(* CODESYS project 底盘控制系统.project

Project tree, tasks and I/O mapping:
  Device : AM521-0808TP/TN, Shenzhen Inovance Control Technology, version 3.5.11.50
      settings: PersistentStartAdddr = 0; PersistentStartEndAddr = 524287; Mode = 1
    application Application
      libraries: Standard, * (System); IoDrvCANopenAxis, 1.11.4.0 (Inovance); HC_CANBus, 0.1.3.0 (Inovance); Util, 3.5.11.0 (System); SM3_Drive_ETC_Inovance, 1.0.5.0 (Inovance); SysFile, * (System); SysTimeRtc, * (System); CmpLog, 3.5.5.0 (System); SysMem, 3.5.5.0 (System); CmpEventMgr, 3.5.8.0 (System); CmpApp, 3.5.11.0 (System); SysTimeCore, * (System)
      task MainTask (cyclic, interval t#4ms, priority 1) calls CANOpen_Task, main
      task CANOPEN (cyclic, interval t#10ms, priority 2) calls nothing
      program main [ST]
      DifferentialMonitor
      program CANOpen_Task [ST]
      global variables GVL
      function block FB_AckermannKinematics [ST]
      trace Trace (task MainTask): main.fbMoveFSD_Torque.FF_Torque_RR, main.fbMoveFSD_Torque.Rr_Target_rpm, main.fbMoveFSD_Torque.Rr_Actual_rpm, main.fbMoveFSD_Torque.SpeedReference, main.fbMoveFSD_Torque.TargetSpeed_kmh, main.fbMoveFSD_Torque.TorqueCmd_RR, main.fbMoveFSD_Torque.Rr_SpeedError, main.fbMoveFSD_Torque.BrakeRequest
      function block FB_SteerPositionPID [ST]
      function block FB_RearWheelVelocityPID [ST]
      function block FB_AckermannInverseKinematics [ST]
      function block FB_UDP [ST]
      function block FB_PWM [ST]
      function block FB_CAN_SCU_1 [ST]
      function block FB_MoveByYaokong [ST]
      function block FB_MoveByFSD [ST]
      function block FB_CAN_CCU [ST]
      function block test [ST]
      function block FB_CAN_VCU_SES_Req [ST]
      function block FB_CAN_BMS [ST]
      function block cantesttest [LD]
      global variables PersistentVars
      function block FB_CAN_MCU_Command [ST]
      function block FB_Depack_MotorStatus2 [ST]
      function block FB_Depack_MotorStatus1 [ST]
      function block FB_MoveControlByTorque_Yaokong [ST]
      function block FB_MoveControlByTorque_FSD [ST]
    ConfigStorage
    Resources List
    Device Diagnosis
    Network Configuration
      LocalBus Config
    HardWare Configuration
    SoftMotion General Axis Pool
    Local Bus
      GL20_2CAN : GL20 2通道CAN通信接口模块, Inovance, order no. 01440308, version 00.00.00.10
          settings: ModuleBaseInfoStruct.BusType = 10; ModuleBaseInfoStruct.RackNumber = 1; ModuleBaseInfoStruct.SlotNumber = 1; COMPort1 = 32; COMPort2 = 33; devGuid1 = 'e5bf4089-cd92-4763-8943-9d7dacf300b6'; devGuid2 = '326b6049-3dfc-42ac-adce-35d035554d5f'
          unmapped channels: RxPDO_CH, TxPDO_CH
    CAN : CAN总线, INOVANCE, version 00.00.00.10
      CAN_Port : CAN Port, Inovance, version 00.00.00.10
          settings: IsFreeCAN = False; DeviceGuid = '83de0e76-e450-4053-a235-86c09473ce3d'; DeviceName = 'GE20_CAN_485'; InterfaceNo = 1; Device = 'AM521-0808TP/TN'; Port = 4; Type = 41108
        CANopen主站 : CANopen主站, Inovance, version 00.00.00.10
            settings: COPManagerSyncStruct.SyncType = 1; COPManagerSyncStruct.SyncPeriod = 10000; COPManagerHeartbeatStruct.Enable = 1; Port NO = 4; IsPortSub = True; IsMainCAN = False; IsCANExt = True; IsLocalCAN = False
          C6049 : CANopen Slaver, Inovance, order no. 1525, version 00.00.00.10
              settings: NodeID = 3; EnableExpertSettings = 1; Error Control.SlaveHeartbeat.ProduceTime = 300; Error Control.SlaveHeartbeat.NrofConsumer = 1; VendorID = 1097; ProductNumber = 1; RevisionNumber = 131075; NrofRxPDO = 4; ValidRxPDO = 2; PdoCommuIndex = 5120; CanId = 515; TxType = 255;  = 1;  = 805306432; PdoCommuIndex = 5121; CanId = 771; TxType = 255;  = 1;  = 805371968; PdoCommuIndex = 5122; CanId = 1027; TxType = 255;  = 1;  = 805437504; PdoCommuIndex = 5123; CanId = 1283; TxType = 255;  = 1;  = 805503040; NrofTxPDO = 4; ValidTxPDO = 3; PdoCommuIndex = 6144; CanId = 387; TxType = 255; InhibitTime = 50;  = 1;  = 805568576; PdoCommuIndex = 6145; CanId = 643; TxType = 255;
                InhibitTime = 50;  = 1;  = 805634112; PdoCommuIndex = 6146; CanId = 899; TxType = 255; InhibitTime = 50;  = 1;  = 805699648; PdoCommuIndex = 6147; CanId = 1155; TxType = 255; InhibitTime = 50;  = 1;  = 805765184; SdoTimeout = 1000; NrofSDO = 31; SdoCommParam = 269877536; SdoErrHandle = 2; SdoJumptoLine = 31; SdoCommParam = 269942800; SdoCommValue = 300; SdoErrHandle = 2; SdoJumptoLine = 31; SdoCommParam = 269746208; SdoCommValue = 2147483779; SdoErrHandle = 2; SdoJumptoLine = 31; SdoCommParam = 269746208; SdoCommValue = 131; SdoErrHandle = 2; SdoJumptoLine = 31; SdoCommParam = 335544608; SdoCommValue = 2147484163; SdoErrHandle = 2; SdoJumptoLine = 31; SdoCommParam = 335610144; SdoCommValue = 2147484419; SdoErrHandle = 2; SdoJumptoLine = 31;
                SdoCommParam = 335610376; SdoCommValue = 255; SdoErrHandle = 2; SdoJumptoLine = 31; SdoCommParam = 369164296; SdoErrHandle = 2; SdoJumptoLine = 31; SdoCommParam = 369164576; SdoCommValue = 805371968; SdoErrHandle = 2; SdoJumptoLine = 31; SdoCommParam = 369164296; SdoCommValue = 1; SdoErrHandle = 2; SdoJumptoLine = 31; SdoCommParam = 335610144; SdoCommValue = 771; SdoErrHandle = 2; SdoJumptoLine = 31; SdoCommParam = 335675680; SdoCommValue = 2147484675; SdoErrHandle = 2; SdoJumptoLine = 31; SdoCommParam = 335741216; SdoCommValue = 2147484931; SdoErrHandle = 2; SdoJumptoLine = 31; SdoCommParam = 402653472; SdoCommValue = 2147484035; SdoErrHandle = 2; SdoJumptoLine = 31; SdoCommParam = 402653704; SdoCommValue = 255; SdoErrHandle = 2; SdoJumptoLine = 31; SdoCommParam = 402653968; SdoCommValue = 50; SdoErrHandle = 2; SdoJumptoLine = 31; SdoCommParam = 402654480;
                SdoErrHandle = 2; SdoJumptoLine = 31; SdoCommParam = 436207624; SdoErrHandle = 2; SdoJumptoLine = 31; SdoCommParam = 436207904; SdoCommValue = 805568576; SdoErrHandle = 2; SdoJumptoLine = 31; SdoCommParam = 436207624; SdoCommValue = 1; SdoErrHandle = 2; SdoJumptoLine = 31; SdoCommParam = 402653472; SdoCommValue = 387; SdoErrHandle = 2; SdoJumptoLine = 31; SdoCommParam = 402719008; SdoCommValue = 2147484291; SdoErrHandle = 2; SdoJumptoLine = 31; SdoCommParam = 402719240; SdoCommValue = 255; SdoErrHandle = 2; SdoJumptoLine = 31; SdoCommParam = 402719504; SdoCommValue = 50; SdoErrHandle = 2; SdoJumptoLine = 31; SdoCommParam = 402720016; SdoErrHandle = 2; SdoJumptoLine = 31; SdoCommParam = 436273160; SdoErrHandle = 2; SdoJumptoLine = 31; SdoCommParam = 436273440; SdoCommValue = 805634112; SdoErrHandle = 2; SdoJumptoLine = 31; SdoCommParam = 436273160;
                SdoCommValue = 1; SdoErrHandle = 2; SdoJumptoLine = 31; SdoCommParam = 402719008; SdoCommValue = 643; SdoErrHandle = 2; SdoJumptoLine = 31; SdoCommParam = 402784544; SdoCommValue = 2147484547; SdoErrHandle = 2; SdoJumptoLine = 31; SdoCommParam = 402850080; SdoCommValue = 2147484803; SdoErrHandle = 2; SdoJumptoLine = 31; FileName = 'C6049.eds'; FileVersion = '0x02'; FileRevision = '0x01'; EDSVersion = '4.0'; Description = 'EDS for 6049  Canopen Slave'; EDS File Path = 'D:\Asoftware\InoProShop\CODESYS\Common\AM600 Data\EdsFile\C6049.eds'; EDSVersion = 'EDLS'; VendorNumber = 1097; ProductName = 'C6049'; ProductNumber = 1; RevisionNumber = 131075; OrderCode = '60'; Baudrate = 368; SimpleBootUpSlave = 1; Granularity = 0; DynamicChannelsSupported = 0; GroupMessaging = 0; NrOfRXPDO = 4; NrOfTXPDO = 4; LSS_Supported = 0; DummyUsage = 0; SDOType = 0; SDOName = 'Set Heartbeat Consumer'; SDOType = 0; SDOName = 'Set Heartbeat Producer';
                SDOType = 0; SDOName = 'Disable Emcy COB-ID'; SDOType = 0; SDOName = 'Set Emcy COB-ID'; SDOType = 0; SDOName = 'Disable PDO'; SDOType = 0; SDOName = 'Disable PDO'; SDOType = 0; SDOName = 'Set transmission type'; SDOType = 0; SDOName = 'Clear PDO mapping'; SDOType = 0; SDOName = 'Set mapping'; SDOType = 0; SDOName = 'Set number of pdos'; SDOType = 0; SDOName = 'Set and enable COB-ID'; SDOType = 0; SDOName = 'Disable PDO'; SDOType = 0; SDOName = 'Disable PDO'; SDOType = 0; SDOName = 'Disable PDO'; SDOType = 0; SDOName = 'Set transmission type'; SDOType = 0; SDOName = 'Set inhibit time'; SDOType = 0; SDOName = 'Set event time'; SDOType = 0; SDOName = 'Clear PDO mapping'; SDOType = 0; SDOName = 'Set mapping'; SDOType = 0; SDOName = 'Set number of pdos'; SDOType = 0; SDOName = 'Set and enable COB-ID'; SDOType = 0; SDOName = 'Disable PDO';
                SDOType = 0; SDOName = 'Set transmission type'; SDOType = 0; SDOName = 'Set inhibit time'; SDOType = 0; SDOName = 'Set event time'; SDOType = 0; SDOName = 'Clear PDO mapping'; SDOType = 0; SDOName = 'Set mapping'; SDOType = 0; SDOName = 'Set number of pdos'; SDOType = 0; SDOName = 'Set and enable COB-ID'; SDOType = 0; SDOName = 'Disable PDO'; SDOType = 0; SDOName = 'Disable PDO'; Recv PDO Mapping Name.Recv PDO Mapping Name = '64 DI0'; Recv PDO Mapping Name.Recv PDO Mapping Name = '64 DI1'; Recv PDO Mapping Name.Recv PDO Mapping Name = '64 AI0'; Recv PDO Mapping Name.Recv PDO Mapping Name = '64 AI1'; Send PDO Mapping Name.Send PDO Mapping Name = '64 DO0'; Send PDO Mapping Name.Send PDO Mapping Name = '64 DO1'; Send PDO Mapping Name.Send PDO Mapping Name = '64 AO0'; Send PDO Mapping Name.Send PDO Mapping Name = '64 AO1'; Is Manual change COB-ID = 0; Is Manual change COB-ID = 0; Is Manual change COB-ID = 0; Is Manual change COB-ID = 0; Is Manual change COB-ID = 0; Is Manual change COB-ID = 0; Is Manual change COB-ID = 0; Is Manual change COB-ID = 0; MandatoryObjs = 3; Object Dictionary Item = '1000;Device Type;0x00000000;7;7;RO;0;-1;-1;-1'; Object Dictionary Item = '1001;Error Register;0x0;5;7;RO;0;-1;-1;-1'; Object Dictionary Item = '1018;Identity Object;;-1;9;;-1;4;-1;-1'; Object Dictionary Item = '1018sub0;number of entries;3;5;7;RO;0;-1;4;1'; Object Dictionary Item = '1018sub1;Vendor ID;0x00000449;7;7;RO;0;-1;-1;-1';
                Object Dictionary Item = '1018sub2;Product code;0x00000001;7;7;RO;0;-1;-1;-1'; Object Dictionary Item = '1018sub3;Revision number;0x00020003;7;7;RO;0;-1;-1;-1'; ManufacturerObjs = 9; Object Dictionary Item = '2000;Index 0x2000;;-1;9;;-1;2;-1;-1'; Object Dictionary Item = '2000sub0;Set TXPDO inhibit time;0x01;5;7;RO;0;-1;-1;-1'; Object Dictionary Item = '2000sub1;TXPDO1 inhibit time;100;5;7;RW;0;-1;-1;-1'; Object Dictionary Item = '3000;64 DI0;0;27;7;RO;1;-1;-1;-1'; Object Dictionary Item = '3001;64 DI1;0x0;27;7;RO;1;-1;-1;-1'; Object Dictionary Item = '3002;64 AI0;0;27;7;RO;1;-1;-1;-1'; Object Dictionary Item = '3003;64 AI1;0x0;27;7;RO;1;-1;-1;-1'; Object Dictionary Item = '3004;64 DO0;0x0;27;7;RWW;1;-1;-1;-1'; Object Dictionary Item = '3005;64 DO1;0x0;27;7;RWW;1;-1;-1;-1'; Object Dictionary Item = '3006;64 AO0;0x0;27;7;RWW;1;-1;-1;-1'; Object Dictionary Item = '3007;64 AO1;0x0;27;7;RWW;1;-1;-1;-1'; OptionsObjs = 20; Object Dictionary Item = '1005;COB-ID SYNC message;0x80;7;7;RW;0;-1;-1;-1'; Object Dictionary Item = '1008;Device Name;4055;9;7;CONST;0;-1;-1;-1'; Object Dictionary Item = '1016;Consumer Heartbeat time group;;-1;8;;-1;2;-1;-1'; Object Dictionary Item = '1016sub0;Number of entries;1;5;7;RO;0;-1;-1;-1'; Object Dictionary Item = '1016sub1;Consumer Heartbeat time;0;7;7;RW;0;-1;-1;-1'; Object Dictionary Item = '1017;Producer Heartbeat time group;0;6;7;RW;0;-1;-1;-1'; Object Dictionary Item = '1400;Receive PDO1 parameter;;-1;9;;-1;4;-1;-1'; Object Dictionary Item = '1400sub0;Number of entries;3;5;7;RO;0;-1;-1;-1'; Object Dictionary Item = '1400sub1;COB-ID;$NodeID + 0x200;7;7;RW;0;-1;-1;-1'; Object Dictionary Item = '1400sub2;Transmission type;255;5;7;RW;0;-1;-1;-1'; Object Dictionary Item = '1400sub3;Inhibit timer;0;5;7;RW;0;-1;-1;-1'; Object Dictionary Item = '1600;Receive PDO1 mapping;;-1;9;;-1;2;-1;-1'; Object Dictionary Item = '1600sub0;Number of mapped objects;0x1;5;7;RO;0;-1;5;0'; Object Dictionary Item = '1600sub1;1.mapped object;0x30000040;7;7;RO;0;-1;-1;-1'; Object Dictionary Item = '1401;Receive PDO2 parameter;;-1;9;;-1;4;-1;-1'; Object Dictionary Item = '1401sub0;Number of entries;3;5;7;RO;0;-1;-1;-1'; Object Dictionary Item = '1401sub1;COB-ID;$NodeID + 0x300;7;7;RW;0;-1;-1;-1'; Object Dictionary Item = '1401sub2;Transmission type;255;5;7;RW;0;-1;-1;-1'; Object Dictionary Item = '1401sub3;Inhibit timer;0;5;7;RW;0;-1;-1;-1'; Object Dictionary Item = '1601;Receive PDO2 mapping;;-1;9;;-1;2;-1;-1'; Object Dictionary Item = '1601sub0;Number of mapped objects;0x1;5;7;RO;0;-1;5;0'; Object Dictionary Item = '1601sub1;1.mapped object;0x30010040;7;7;RO;0;-1;-1;-1'; Object Dictionary Item = '1402;Receive PDO3 parameter;;-1;9;;-1;4;-1;-1'; Object Dictionary Item = '1402sub0;Number of entries;3;5;7;RO;0;-1;-1;-1'; Object Dictionary Item = '1402sub1;COB-ID;$NodeID + 0x400;7;7;RW;0;-1;-1;-1';
                Object Dictionary Item = '1402sub2;Transmission type;255;5;7;RW;0;-1;-1;-1'; Object Dictionary Item = '1402sub3;Inhibit timer;0;5;7;RW;0;-1;-1;-1'; Object Dictionary Item = '1602;Receive PDO3 mapping;;-1;9;;-1;2;-1;-1'; Object Dictionary Item = '1602sub0;Number of mapped objects;0x1;5;7;RO;0;-1;5;0'; Object Dictionary Item = '1602sub1;1.mapped object;0x30020040;7;7;RO;0;-1;-1;-1'; Object Dictionary Item = '1403;Receive PDO4 parameter;;-1;9;;-1;4;-1;-1'; Object Dictionary Item = '1403sub0;Number of entries;3;5;7;RO;0;-1;-1;-1'; Object Dictionary Item = '1403sub1;COB-ID;$NodeID + 0x500;7;7;RW;0;-1;-1;-1'; Object Dictionary Item = '1403sub2;Transmission type;255;5;7;RW;0;-1;-1;-1'; Object Dictionary Item = '1403sub3;Inhibit timer;0;5;7;RW;0;-1;-1;-1'; Object Dictionary Item = '1603;Receive PDO4 mapping;;-1;9;;-1;2;-1;-1'; Object Dictionary Item = '1603sub0;Number of mapped objects;0x1;5;7;RO;0;-1;5;0'; Object Dictionary Item = '1603sub1;1.mapped object;0x30030040;7;7;RO;0;-1;-1;-1'; Object Dictionary Item = '1800;Transmit PDO1 parameter;;-1;9;;-1;5;-1;-1'; Object Dictionary Item = '1800sub0;Number of entries;0x5;5;7;RO;0;-1;-1;-1'; Object Dictionary Item = '1800sub1;COB-ID;$NodeID + 0x180;7;7;RW;0;-1;-1;-1'; Object Dictionary Item = '1800sub2;Transmission type;255;5;7;RW;0;-1;-1;-1'; Object Dictionary Item = '1800sub3;Inhibit timer;50;6;7;RW;0;-1;-1;-1'; Object Dictionary Item = '1800sub5;Event Timer;0;27;7;RW;0;-1;65535;0'; Object Dictionary Item = '1A00;Transmit PDO1 mapping;;-1;9;;-1;2;-1;-1'; Object Dictionary Item = '1A00sub0;Number of mapped objects;0x1;5;7;RO;0;-1;4;0'; Object Dictionary Item = '1A00sub1;1.mapped object;0x30040040;7;7;RO;0;-1;-1;-1'; Object Dictionary Item = '1801;Transmit PDO2 parameter;;-1;9;;-1;5;-1;-1'; Object Dictionary Item = '1801sub0;Number of entries;0x5;5;7;RO;0;-1;-1;-1'; Object Dictionary Item = '1801sub1;COB-ID;$NodeID + 0x280;7;7;RW;0;-1;-1;-1'; Object Dictionary Item = '1801sub2;Transmission type;255;5;7;RW;0;-1;-1;-1'; Object Dictionary Item = '1801sub3;Inhibit timer;50;6;7;RW;0;-1;-1;-1'; Object Dictionary Item = '1801sub5;Event Timer;0;27;7;RW;0;-1;65535;0'; Object Dictionary Item = '1A01;Transmit PDO2 mapping;;-1;9;;-1;2;-1;-1'; Object Dictionary Item = '1A01sub0;Number of mapped objects;0x1;5;7;RO;0;-1;4;0'; Object Dictionary Item = '1A01sub1;1.mapped object;0x30050040;7;7;RO;0;-1;-1;-1'; Object Dictionary Item = '1802;Transmit PDO3 parameter;;-1;9;;-1;5;-1;-1'; Object Dictionary Item = '1802sub0;Number of entries;0x5;5;7;RO;0;-1;-1;-1'; Object Dictionary Item = '1802sub1;COB-ID;$NodeID + 0x380;7;7;RW;0;-1;-1;-1'; Object Dictionary Item = '1802sub2;Transmission type;255;5;7;RW;0;-1;-1;-1'; Object Dictionary Item = '1802sub3;Inhibit timer;50;6;7;RW;0;-1;-1;-1'; Object Dictionary Item = '1802sub5;Event Timer;0;27;7;RW;0;-1;65535;0'; Object Dictionary Item = '1A02;Transmit PDO3 mapping;;-1;9;;-1;2;-1;-1'; Object Dictionary Item = '1A02sub0;Number of mapped objects;0x1;5;7;RO;0;-1;4;0'; Object Dictionary Item = '1A02sub1;1.mapped object;0x30060040;7;7;RO;0;-1;-1;-1';
                Object Dictionary Item = '1803;Transmit PDO4 parameter;;-1;9;;-1;5;-1;-1'; Object Dictionary Item = '1803sub0;Number of entries;0x5;5;7;RO;0;-1;-1;-1'; Object Dictionary Item = '1803sub1;COB-ID;$NodeID + 0x480;7;7;RW;0;-1;-1;-1'; Object Dictionary Item = '1803sub2;Transmission type;255;5;7;RW;0;-1;-1;-1'; Object Dictionary Item = '1803sub3;Inhibit timer;50;6;7;RW;0;-1;-1;-1'; Object Dictionary Item = '1803sub5;Event Timer;0;27;7;RW;0;-1;65535;0'; Object Dictionary Item = '1A03;Transmit PDO4 mapping;;-1;9;;-1;2;-1;-1'; Object Dictionary Item = '1A03sub0;Number of mapped objects;0x1;5;7;RO;0;-1;4;0'; Object Dictionary Item = '1A03sub1;1.mapped object;0x30070040;7;7;RO;0;-1;-1;-1'
              output Application.YkqRxPDO0_data : LWORD  // 64 DI1
              input  Application.YkqTxPDO0_data : LWORD  // 64 DO0
              input  Application.Emergency_Stop : BOOL  // 64 DO0.Bit0
              input  Application.DriveByYaokong : BOOL  // 64 DO0.Bit10
              input  Application.DriveBySelf : BOOL  // 64 DO0.Bit11
              input  Application.Remote_Break : BOOL  // 64 DO0.Bit15
              input  Application.YkqTxPDO1_data : LWORD  // 64 DO1
      CAN_Port_1 : CAN Port, Inovance, version 00.00.00.10
          settings: IsFreeCAN = True; DeviceGuid = '41b44ff1-ebbe-4db4-bb20-eb005c34d964'; DeviceName = 'GL20_2CAN'; Port = 32; Type = 41090
        CAN自由协议 : CAN自由协议, Inovance, version 00.00.00.10
            settings: CANBusGeneralStruct.BusNodeID = 32; IsPortSub = True; IsLocalCAN = True; IsFreeCAN = True; DeviceTaskName = 'MainTask'; IsVirtual = True; VirtualInterface = 0; TotalChannelCount = 7; channel0.SendingMethod = False; channel0.FrameType = False; channel0.FrameFormat = False; channel0.FrameID = 361; channel0.NumberOfBytes = 8; channel0.RetransmissionInterval = 20; channel0.CycleSendingTime = 20; channel0.IOMappingParamId = 4285874176; channel1.uiChannelIndex = 1; channel1.SendingMethod = False; channel1.FrameType = False; channel1.FrameFormat = False; channel1.FrameID = 617; channel1.NumberOfBytes = 8; channel1.RetransmissionInterval = 20; channel1.CycleSendingTime = 20; channel1.IOMappingParamId = 4285874177; channel2.uiChannelIndex = 2; channel2.SendingMethod = False; channel2.FrameType = False; channel2.FrameFormat = False; channel2.FrameID = 1977; channel2.NumberOfBytes = 8; channel2.RetransmissionInterval = 5; channel2.CycleSendingTime = 10; channel2.IOMappingParamId = 4285874178; channel3.uiChannelIndex = 3; channel3.SendingMethod = False; channel3.FrameType = False; channel3.FrameFormat = False; channel3.FrameID = 256; channel3.NumberOfBytes = 8;
              channel3.RetransmissionInterval = 5; channel3.CycleSendingTime = 10; channel3.IOMappingParamId = 4285874179; channel4.uiChannelIndex = 4; channel4.SendingMethod = False; channel4.FrameType = False; channel4.FrameFormat = False; channel4.FrameID = 81; channel4.NumberOfBytes = 8; channel4.RetransmissionInterval = 5; channel4.CycleSendingTime = 10; channel4.IOMappingParamId = 4285874180; channel5.uiChannelIndex = 5; channel5.SendingMethod = False; channel5.FrameType = True; channel5.FrameFormat = False; channel5.FrameID = 285206679; channel5.NumberOfBytes = 8; channel5.RetransmissionInterval = 5; channel5.CycleSendingTime = 20; channel5.IOMappingParamId = 4285874181; channel6.uiChannelIndex = 6; channel6.SendingMethod = False; channel6.FrameType = True; channel6.FrameFormat = False; channel6.FrameID = 285205911; channel6.NumberOfBytes = 8; channel6.RetransmissionInterval = 5; channel6.CycleSendingTime = 10; channel6.IOMappingParamId = 4285874182
            input  Application.ReciveCanID : DWORD  // Receive Data.FrameID
            input  Application.ReciveCanData  // Receive Data.FrameFirstAddressArray
            output Application.CAN_SES_Req_Data_F : ARRAY [0..7] OF BYTE  // Channel0
            output Application.CAN_SES_Req_Data_R : ARRAY [0..7] OF BYTE  // Channel1
            output Application.VCU_SEB_Req_Data : ARRAY [0..7] OF BYTE  // Channel2
            output Application.main.fbMoveFSD_Torque.BMS_Send_Data : ARRAY [0..7] OF BYTE  // Channel3
            output Application.main.fbMoveFSD_Torque.CCU_CAN_Data : ARRAY [0..7] OF BYTE  // Channel4
            output Application.CAN_Motor_Cmd_RR : ARRAY [0..7] OF BYTE  // Channel5
            output Application.CAN_Motor_Cmd_RL : ARRAY [0..7] OF BYTE  // Channel6
            unmapped channels: Receive Data
      CAN_Port_2 : CAN Port, Inovance, version 00.00.00.10
          settings: IsFreeCAN = False; DeviceGuid = '41b44ff1-ebbe-4db4-bb20-eb005c34d964'; DeviceName = 'GL20_2CAN'; InterfaceNo = 1; Port = 33; Type = 41090
    Serial : 串行接口, 汇川技术股份有限公司, version 00.00.00.10
      COM : Serial Port, Inovance, version 00.00.00.10
          settings: Device = AM521-0808TP/TN; devGuid = 'e348f94f-2bae-4e83-9430-22bd03696b88'
      COM_1 : Serial Port, Inovance, version 00.00.00.10
          settings: COM = 4; Device = GE20_CAN_485; Type = 1; devGuid = '83de0e76-e450-4053-a235-86c09473ce3d'
    LocalHSIO : 本地高速IO, 汇川技术股份有限公司, version 2.0.0.0
        input  Application.IsCollisionF : BOOL  // DigitalInput.Bit0
        input  Application.IsCollisionR : BOOL  // DigitalInput.Bit1
        output Application.PDO_IO_Output0 : BOOL  // DigitalOutput.Bit0
        output Application.PDO_IO_Output1 : BOOL  // DigitalOutput.Bit1
        unmapped channels: DigitalInput, DigitalOutput
    EXP_A : 扩展卡, 汇川技术股份有限公司, version 00.00.00.10
      GE20_CAN_485 : GE20_CAN_485, Inovance, version 1.0.0.0
          settings: GE20_CAN_485 ExtCard configure.SerialAlias = 4; GE20_CAN_485 ExtCard configure.CANAlias = 4
    EXP_B : 扩展卡, 汇川技术股份有限公司, version 00.00.00.10
    HwConfiguratioinDevice : SystemConfig, Inovance, version 00.00.00.10
        settings: NetworkConfigArray.NetworkConfigArray.BusType = 10; NetworkConfigArray.NetworkConfigArray.RackSum = 1; NetworkConfigArray.NetworkConfigArray.HardwareConfigArray.HardwareConfigArray.RackNo = 1; NetworkConfigArray.NetworkConfigArray.HardwareConfigArray.HardwareConfigArray.ModuleNum = 1; EnableFun = 1
*)

// Device/Application/GVL
VAR_GLOBAL
	//遥控器参数接收
	YkqTxPDO0_data	:	ARRAY[0..7] OF BYTE;
	YkqTxPDO1_data	:	ARRAY[0..7] OF BYTE;
	YkqRxPDO0_data	:	ARRAY[0..7] OF BYTE;
	DriveBySelf		:	BOOL ;
	DriveByYaokong	:	BOOL ;
	Emergency_Stop	:	BOOL;
	Remote_Break	:	BOOL;
	
	
	

	//PDO 写入的相关数据
	//电机实际转速
    ActVel_RPM_RL   : DINT; (*  (rpm) *)
    ActVel_RPM_RR   : DINT; (*  (rpm) *)

	
	// 转向系统
     CAN_SES_Req_R : FB_CAN_VCU_SES_Req;
     CAN_SES_Req_F : FB_CAN_VCU_SES_Req;
	 CAN_SES_Req_Data_F : ARRAY[0..7] OF BYTE;
     CAN_SES_Req_Data_R : ARRAY[0..7] OF BYTE;
	 //制动系统
	 VCU_SEB_Req_Data : ARRAY[0..7] OF BYTE;
	 
	 //触边检测
	 IsCollisionF	: BOOL := FALSE;
	 IsCollisionR	: BOOL := FALSE;
	 
	 //云乐电机控制指令
	 //电机左后轮 驱动电机，CAN通道6  	 ID 10FFE597  十进制285205911
	 //电机右后轮 转向电机，CAN通道5	 ID 10FFE897  十进制285206679
	 CAN_Motor_Cmd_RR	:	ARRAY[0..7] OF BYTE;
	 CAN_Motor_Cmd_RL	:	ARRAY[0..7] OF BYTE;
	 //GCAN 212发送数据（电机指令）
	 GCAN212_Send_RR_cmd     : ARRAY[0..12] OF BYTE;
	 GCAN212_Send_RL_cmd     : ARRAY[0..12] OF BYTE;
	 GCAN212_Recive_RR_status1 : ARRAY[0..7] OF BYTE;
	 GCAN212_Recive_RR_status2 : ARRAY[0..7] OF BYTE;
	 GCAN212_Recive_RL_status1 : ARRAY[0..7] OF BYTE;
	 GCAN212_Recive_RL_status2 : ARRAY[0..7] OF BYTE;
	 
	 //自动驾驶发送控制指令，通过UDP接收
	 UDP_Re_FSD_Cmd	:	ARRAY[0..12] OF BYTE;
	 
	 
	//单、双阿克曼切换标志
	//True 是单阿克曼、FALSE是双阿克曼
	AckermanModleTransfer	:	BOOL;
	
	//CAN 总线收到的数据
	ReciveCanData	:	ARRAY[0..7] OF BYTE;
	ReciveCanID		:	DWORD;
	
	//PDO，IO信号处理，防撞条一侧为True
	PDO_IO_Output0	:	BOOL	:= TRUE;
	PDO_IO_Output1	:	BOOL	:= TRUE;
	

END_VAR

// Device/Application/PersistentVars
{attribute 'qualified_only'}
VAR_GLOBAL PERSISTENT RETAIN
END_VAR

// Device/Application/CANOpen_Task
PROGRAM CANOpen_Task
VAR
END_VAR

END_PROGRAM

// Device/Application/main
PROGRAM main
VAR

	
	fbUdp		: FB_UDP;

	fbMoveYkq	: FB_MoveByYaokong;
	fbMoveFSD	: FB_MoveByFSD;
	fbMoveYkq_Torque	:	FB_MoveControlByTorque_Yaokong;
	fbMoveFSD_Torque	:	FB_MoveControlByTorque_FSD;
	
	recvBuf     : ARRAY[0..12] OF BYTE;
	
	

	
END_VAR






fbUdp();
IF DriveBySelf THEN	
	//fbMoveFSD();
	fbMoveFSD_Torque();
	
ELSIF DriveByYaokong THEN
	//遥控器控制
	//fbMoveYkq();
	fbMoveYkq_Torque();
END_IF

END_PROGRAM

// Device/Application/FB_UDP
FUNCTION_BLOCK FB_UDP
VAR_INPUT
	//xEnable     : BOOL;               // 是否使能工作
	//sendBuf_RR_Motor_Cmd	 	: ARRAY[0..12] OF BYTE;
	//sendBuf_RL_Motor_Cmd	 	: ARRAY[0..12] OF BYTE;
END_VAR
VAR_OUTPUT
	//recvBuf     : ARRAY[0..12] OF BYTE;
	
	
END_VAR
VAR
	UDP_Peer_RR	:	UDP_Peer;
	UDP_Peer_RL	:	UDP_Peer;
	UDP_Peer_FSD	:	UDP_Peer;

	UDP_Send_RR_Motor_Cmd	:	UDP_Send;
	UDP_Send_RL_Motor_Cmd	:	UDP_Send;
	UDP_Receive_RR	:	UDP_Receive;
	UDP_Receive_RL	:	UDP_Receive;
	UDP_Receive_FSD	:	UDP_Receive;
	
	IpAddrLocal_RR	:	STRING	:= '192.168.100.210';
	PortLocal_RR	:	UINT	:= 5001;
	hPeer_RR		:	DWORD;
	IpAddrLocal_RL	:	STRING	:= '192.168.100.210';
	PortLocal_RL	:	UINT	:= 5002;
	hPeer_RL		:	DWORD;
	IpAddrLocal_FSD	:	STRING	:= '192.168.100.210';
	PortLocal_FSD	:	UINT	:= 5003;
	hPeer_FSD		:	DWORD;
	
	remoteIP_RR_Motor    : STRING(80) := '192.168.100.20';
	remotePort_RR_Motor  : UINT := 4001;
	remoteIP_RL_Motor    : STRING(80) := '192.168.100.20';
	remotePort_RL_Motor  : UINT := 4002;

	
	recvbuf_RR	: ARRAY[0..12] OF BYTE;
	recvbuf_RL	: ARRAY[0..12] OF BYTE;
	recvbuf_FSD	: ARRAY[0..12] OF BYTE;
	
	CanID_RR	: UDINT;
	CanID_RL	: UDINT;


	SendErrorID_RR		:	DWORD;
	SendErrorID_RL		:	DWORD;
	bSendDone_RR		:	BOOL;
	bSendDone_RL		:	BOOL;
	bSendBusy_RR		:	BOOL;
	bSendBusy_RL		:	BOOL;
	bRecvDone_RR 		:	BOOL;
    bRecvBusy_RR 		:	BOOL;
    bRecvDone_RL 		:	BOOL;
    bRecvBusy_RL 		:	BOOL;

	

	
	fbPWM	:	FB_PWM;
	pwm	:	BOOL;
	//rTrigSend : R_TRIG;
	PeerErrorID_RR: DWORD;
	PeerErrorID_RL: DWORD;
	
	 rTrigRecv   : R_TRIG;
	 (*-------------通信超时-------------*)
    udiLastRecvTime : UDINT := 0;      // 上一次收到UDP数据时间(ms)
    udiNowTime      : UDINT;           // 当前时间(ms)
END_VAR


// ***********RR电机*********
UDP_Peer_RR(
	xEnable:=TRUE,
	strIpAddrLocal:=IpAddrLocal_RR,
	uiPortLocal:=PortLocal_RR,
	dwErrorID =>PeerErrorID_RR);

hPeer_RR := UDP_Peer_RR.hPeer;

UDP_Receive_RR(xEnable:=TRUE,
		hPeer := hPeer_RR,
		uiSize := SIZEOF(recvbuf_RR),
		pbyData := ADR(recvbuf_RR),
		xBusy => bRecvBusy_RR,
		xDone => bRecvDone_RR
		);
		
// **********RL电机***********
UDP_Peer_RL(
	xEnable:=TRUE,
	strIpAddrLocal:=IpAddrLocal_RL,
	uiPortLocal:=PortLocal_RL,
	dwErrorID =>PeerErrorID_RL);

hPeer_RL := UDP_Peer_RL.hPeer;
UDP_Receive_RL(xEnable:=TRUE,
		hPeer := hPeer_RL,
		uiSize := SIZEOF(recvbuf_RL),
		pbyData := ADR(recvbuf_RL),
		xBusy => bRecvBusy_RL,
		xDone => bRecvDone_RL
		);

//**********接收智驾控制信号**********
UDP_Peer_FSD(
	xEnable:=TRUE,
	strIpAddrLocal:=IpAddrLocal_FSD,
	uiPortLocal:=PortLocal_FSD);
	
hPeer_FSD := UDP_Peer_FSD.hPeer;

UDP_Receive_FSD(xEnable:=TRUE,
		hPeer := hPeer_FSD,
		uiSize := SIZEOF(recvbuf_FSD),
		pbyData := ADR(recvbuf_FSD)
		);



CanID_RR :=
    SHL(BYTE_TO_UDINT(recvbuf_RR[1]),24) OR
    SHL(BYTE_TO_UDINT(recvbuf_RR[2]),16) OR
    SHL(BYTE_TO_UDINT(recvbuf_RR[3]),8)  OR
         BYTE_TO_UDINT(recvbuf_RR[4]);
CanID_RL :=
    SHL(BYTE_TO_UDINT(recvbuf_RL[1]),24) OR
    SHL(BYTE_TO_UDINT(recvbuf_RL[2]),16) OR
    SHL(BYTE_TO_UDINT(recvbuf_RL[3]),8)  OR
         BYTE_TO_UDINT(recvbuf_RL[4]);


IF CanID_RR = 16#18FFE699 THEN
	GVL.GCAN212_Recive_RR_status1[0] := recvbuf_RR[5];
    GVL.GCAN212_Recive_RR_status1[1] := recvbuf_RR[6];
    GVL.GCAN212_Recive_RR_status1[2] := recvbuf_RR[7];
    GVL.GCAN212_Recive_RR_status1[3] := recvbuf_RR[8];
    GVL.GCAN212_Recive_RR_status1[4] := recvbuf_RR[9];
    GVL.GCAN212_Recive_RR_status1[5] := recvbuf_RR[10];
    GVL.GCAN212_Recive_RR_status1[6] := recvbuf_RR[11];
    GVL.GCAN212_Recive_RR_status1[7] := recvbuf_RR[12];
ELSIF CanID_RR = 16#18FFE799 THEN
	GVL.GCAN212_Recive_RR_status2[0] := recvbuf_RR[5];
    GVL.GCAN212_Recive_RR_status2[1] := recvbuf_RR[6];
    GVL.GCAN212_Recive_RR_status2[2] := recvbuf_RR[7];
    GVL.GCAN212_Recive_RR_status2[3] := recvbuf_RR[8];
    GVL.GCAN212_Recive_RR_status2[4] := recvbuf_RR[9];
    GVL.GCAN212_Recive_RR_status2[5] := recvbuf_RR[10];
    GVL.GCAN212_Recive_RR_status2[6] := recvbuf_RR[11];
    GVL.GCAN212_Recive_RR_status2[7] := recvbuf_RR[12];
END_IF

IF CanID_RL = 16#18FFE699 THEN
	GVL.GCAN212_Recive_RL_status1[0] := recvbuf_RL[5];
    GVL.GCAN212_Recive_RL_status1[1] := recvbuf_RL[6];
    GVL.GCAN212_Recive_RL_status1[2] := recvbuf_RL[7];
    GVL.GCAN212_Recive_RL_status1[3] := recvbuf_RL[8];
    GVL.GCAN212_Recive_RL_status1[4] := recvbuf_RL[9];
    GVL.GCAN212_Recive_RL_status1[5] := recvbuf_RL[10];
    GVL.GCAN212_Recive_RL_status1[6] := recvbuf_RL[11];
    GVL.GCAN212_Recive_RL_status1[7] := recvbuf_RL[12];
ELSIF CanID_RL = 16#18FFE799 THEN
	GVL.GCAN212_Recive_RL_status2[0] := recvbuf_RL[5];
    GVL.GCAN212_Recive_RL_status2[1] := recvbuf_RL[6];
    GVL.GCAN212_Recive_RL_status2[2] := recvbuf_RL[7];
    GVL.GCAN212_Recive_RL_status2[3] := recvbuf_RL[8];
    GVL.GCAN212_Recive_RL_status2[4] := recvbuf_RL[9];
    GVL.GCAN212_Recive_RL_status2[5] := recvbuf_RL[10];
    GVL.GCAN212_Recive_RL_status2[6] := recvbuf_RL[11];
    GVL.GCAN212_Recive_RL_status2[7] := recvbuf_RL[12];
END_IF

//将接受到的智驾数据转到全局变量，便于FSD程序调用
GVL.UDP_Re_FSD_Cmd := recvbuf_FSD;

		
//发送
fbPWM(Enable:=TRUE,HalfPeriod:=T#10MS);
pwm := fbPWM.PWM;
	
UDP_Send_RR_Motor_Cmd(xExecute:=pwm,
	hPeer := hPeer_RR,
	strIpAddrDst := remoteIP_RR_Motor,
	uiPortDst := remotePort_RR_Motor,
	uiSize := SIZEOF(GVL.GCAN212_Send_RR_cmd),
	pbyData := ADR(GVL.GCAN212_Send_RR_cmd),
	udiTimeOut:=500000,
	dwErrorID => SendErrorID_RR,
	xDone	=>	bSendDone_RR,
	xBusy	=>	bSendBusy_RR
);	
UDP_Send_RL_Motor_Cmd(xExecute:=pwm,
	hPeer := hPeer_RL,
	strIpAddrDst := remoteIP_RL_Motor,
	uiPortDst := remotePort_RL_Motor,
	uiSize := SIZEOF(GVL.GCAN212_Send_RL_cmd),
	pbyData := ADR(GVL.GCAN212_Send_RL_cmd),
	udiTimeOut:=500000,
	dwErrorID => SendErrorID_RL,
	xDone	=>	bSendDone_RL,
	xBusy	=>	bSendBusy_RL
);	

(*******************************)
(* UDP通信超时检测             *)
(*******************************)

END_FUNCTION_BLOCK

// Device/Application/FB_PWM
FUNCTION_BLOCK FB_PWM
VAR_INPUT
	Enable     : BOOL := TRUE;        // 使能输出
    HalfPeriod : TIME ;     // 半周期（默认500ms -> 总周期1s）
END_VAR
VAR_OUTPUT
	PWM        : BOOL := FALSE;       // 输出的PWM布尔量
END_VAR
VAR
	tmr : TON;                        // 定时器（标准TON）
END_VAR

IF NOT Enable THEN
    PWM := FALSE;
    tmr(IN := FALSE);    // 停止并复位定时器
ELSE
    // 定时器启动：计时到达 HalfPeriod 时 tmr.Q = TRUE
    tmr(IN := TRUE, PT := HalfPeriod);

    IF tmr.Q THEN
        // 到达半周期：翻转PWM并复位定时器以开始下一半周期
        PWM := NOT PWM;
        tmr(IN := FALSE);    // 复位定时器（下一循环会再设为 TRUE 重启计时）
    END_IF
END_IF

END_FUNCTION_BLOCK

// Device/Application/FB_MoveByYaokong
(*
====================================================================
 FB 名称 : FB_MoveByYaokong
 功能说明 :
 1. 解析遥控器 CAN 数据
 2. 计算目标车速与转向角
 3. Ackermann 底盘运动学解算
 4. 转向 CAN 报文下发
 5. 驱动轮速度控制
 6. 急停 / 驻车逻辑
 7. 车辆状态回传
====================================================================
*)

FUNCTION_BLOCK FB_MoveByYaokong

//====================================================================
// 输入输出
//====================================================================
VAR_INPUT
END_VAR

VAR_OUTPUT
END_VAR


//====================================================================
// 遥控器输入相关
//====================================================================
VAR
	
	fbMotorCmd_RR		:	FB_CAN_MCU_Command;
	fbMotorCmd_RL		:	FB_CAN_MCU_Command;
    // 遥控器原始数据
    RemoteDriveRaw    : BYTE;     // 前后拨杆
    RemoteSteerRaw    : BYTE;     // 左右拨杆

    // 遥控器中位与死区
    DriveCenter       : INT := 16#7F;
    DriveDeadband     : INT := 5;

    // 遥控器解析变量
    DriveOffset       : INT;
    DriveRatio        : LREAL;
    SteeringRatio     : REAL;

    // 方向标志
    Dir_FR            : BYTE;     // 前后方向
    Dir_LR            : BYTE;     // 左右方向
END_VAR


//====================================================================
// 车辆运动控制相关
//====================================================================
VAR
    // 目标速度
    TargetSpeedMax_kmh : LREAL;
    TargetSpeed_kmh    : LREAL;
	TargetSpeed_kmhtest: LREAL;
	
    // 电机目标转速
    Rr_Speed_rpm       : LREAL;
    Rl_Speed_rpm       : LREAL;
	//电机使能标志 刹车时不使能电机
	Enable_Motor	:	BOOL  := TRUE;
	//车辆行驶档位  0:N  1:D  2:R
	RR_Shift_leavel	:	BYTE;   
	RL_Shift_leavel	:	BYTE;
	//电机驱动方式  1:速度  0:力矩
	Motor_Drive_mode_RR	:	BOOL := 1 ;
	Motor_Drive_mode_RL	:	BOOL := 1 ;
	
    // 转向角
    SteeringDeg        : REAL;
    SteeringRad        : REAL;
	
	//电机状态解包
	fbDepack_MotorStatus1_RR	:	FB_Depack_MotorStatus1;
	fbDepack_MotorStatus2_RR	:	FB_Depack_MotorStatus2;
	fbDepack_MotorStatus1_RL	:	FB_Depack_MotorStatus1;
	fbDepack_MotorStatus2_RL	:	FB_Depack_MotorStatus2;
END_VAR


//====================================================================
// 转向机构参数
//====================================================================
VAR
    // 转向机构参数
    Ls_mm              : REAL := 100.0;     // 转向节转臂长度
    Pitch_mm           : REAL := 43.692;    // 转向器线角比

    // 转向计算中间量
    RackTravel_mm      : REAL;
    SteerAngle_deg     : REAL;

    // 常量
    PI                 : REAL := 3.1415926;
END_VAR


//====================================================================
// 运动学功能块
//====================================================================
VAR
    fbKine             : FB_AckermannKinematics;
    fbInvKine          : FB_AckermannInverseKinematics;
END_VAR


//====================================================================
// 驱动器控制功能块
//====================================================================
VAR
    // 右后轮
    fbPower_RR         : MC_Power_CO;
    fbMoveVel_RR       : MC_MoveVelocity_CO;
    fbStop_RR          : MC_Stop_CO;

    // 左后轮
    fbPower_RL         : MC_Power_CO;
    fbMoveVel_RL       : MC_MoveVelocity_CO;
    fbStop_RL          : MC_Stop_CO;
END_VAR


//====================================================================
// Execute脉冲控制
//====================================================================
VAR
    // 上一次速度记录
    PreSpeed_RR        : LREAL := 0.0;
    PreSpeed_RL        : LREAL := 0.0;

    // 速度变化检测
    SpeedChanged_RR    : BOOL;
    SpeedChanged_RL    : BOOL;

    // Execute脉冲
    ExecuteMove_RR     : BOOL := FALSE;
    ExecuteMove_RL     : BOOL := FALSE;

    // 单周期保持
    PulseHold_RR       : BOOL := FALSE;
    PulseHold_RL       : BOOL := FALSE;
END_VAR


//====================================================================
// 制动与驻车系统
//====================================================================
VAR
    ParkingButton      : BOOL := FALSE;
    ParkingState       : BOOL := FALSE;

    PressureValue      : BYTE := 0;
	BrakeRequest       : BOOL := FALSE;   //<<<< 新增统一刹车请求
    rTrigBtn           : R_TRIG;
END_VAR

//====================================================================
// 电机状态反馈 UDP接收到的
//====================================================================
VAR
	RR_Motor_CanID : UDINT;
	RL_Motor_CanID : UDINT;
	
END_VAR

//====================================================================
// 减速控制
//====================================================================
VAR
	// 当前是否减速
	RR_Decelerating : BOOL;
	RL_Decelerating : BOOL;
	//速度差 = 实际速度 - 目标速度
	RR_SpeedError : REAL;
    RL_SpeedError : REAL;
	// P控制
	BrakeKp : REAL := 3;      // Nm/rpm
	
	// 最大制动力矩
	BrakeTorqueMax : REAL := 130;
	
	// 当前扭矩
	RR_BrakeTorque : REAL;
	RL_BrakeTorque : REAL;
	
	// 发送给驱动器
	RR_TorqueCmd : INT;
	RR_TorqueCmd_test : INT := -30;
	RL_TorqueCmd : INT;
	
END_VAR

//====================================================================
// 其他状态变量
//====================================================================
VAR
    Break              : BOOL := FALSE;
END_VAR

(*
====================================================================
 1. 遥控器输入解析
====================================================================
*)

TargetSpeedMax_kmh := BYTE_TO_LREAL(YkqTxPDO1_data[0]) / 10.0;


RemoteDriveRaw := YkqTxPDO1_data[1];
RemoteSteerRaw := YkqTxPDO1_data[2];

Dir_FR := RemoteDriveRaw;


(*
====================================================================
 2. 前后拨杆 -> 速度比例计算
====================================================================
*)

DriveOffset := BYTE_TO_INT(RemoteDriveRaw) - DriveCenter;

// 死区处理
IF ABS(DriveOffset) <= DriveDeadband THEN

    DriveRatio := 0.0;

ELSE

    DriveRatio :=
        INT_TO_LREAL(ABS(DriveOffset) - DriveDeadband) /
        INT_TO_LREAL(127 - DriveDeadband);

END_IF;


// 限幅
IF DriveRatio > 1.0 THEN

    DriveRatio := 1.0;

ELSIF DriveRatio < 0.0 THEN

    DriveRatio := 0.0;

END_IF;


// 最终目标速度
TargetSpeed_kmh := TargetSpeedMax_kmh * DriveRatio;

//测试
//TargetSpeed_kmh:=TargetSpeed_kmhtest;

(*
====================================================================
 3. 左右拨杆 -> 转向角计算
====================================================================
*)

// 转向方向
IF RemoteSteerRaw < 127 THEN
    Dir_LR := 1;
ELSE
    Dir_LR := 2;
END_IF;


// 比例映射
SteeringRatio := BYTE_TO_REAL(RemoteSteerRaw) / 255.0;


// 映射到车轮转角
SteeringDeg := -20.0 + (SteeringRatio * 40.0);

// //测试写死
// SteeringDeg	:= 5;
// TargetSpeed_kmh	:= 5;

// 角度 -> 弧度
SteeringRad := SteeringDeg * PI / 180.0;



(*
====================================================================
 4. 转向机构解算
====================================================================
*)

// 轮胎转角 -> 齿条位移
RackTravel_mm := Ls_mm * SteeringRad;


// 齿条位移 -> 转向电机角度
SteerAngle_deg := (RackTravel_mm / Pitch_mm) * 360.0;



(*
====================================================================
 5. 转向 CAN 报文下发
====================================================================
*)

// 前桥转向
CAN_SES_Req_F(
    Tgt_StrAngle    := SteerAngle_deg,
    Tgt_StrAngleSpd := 200,
    Veh_Spd         := 50,
    Enable          := 1
);

CAN_SES_Req_Data_F := CAN_SES_Req_F.CanData;


// 后桥转向（反向）
CAN_SES_Req_R(
    Tgt_StrAngle    := -SteerAngle_deg,
    Tgt_StrAngleSpd := 200,
    Veh_Spd         := 50,
    Enable          := 1
);

CAN_SES_Req_Data_R := CAN_SES_Req_R.CanData;



(*
====================================================================
 6. Ackermann运动学解算
====================================================================
*)

fbKine(
    v_kmh := TargetSpeed_kmh,
    delta := SteeringRad,
    Dir_LR := Dir_LR
);


// 输出轮速
Rr_Speed_rpm :=  fbKine.wRR_rpm;
Rl_Speed_rpm :=  fbKine.wRL_rpm;     // 左右电机对向安装

(*
====================================================================
 7. 行驶方向处理
====================================================================
*)
//清空刹车请求
BrakeRequest := FALSE;

IF DriveRatio < 0.0 THEN

    Rr_Speed_rpm := 0.0;
    Rl_Speed_rpm := 0.0;

    BrakeRequest := TRUE;

ELSIF DriveOffset > 0 THEN

    RR_Shift_leavel := 2;
    RL_Shift_leavel := 1;
	//RR_SpeedError := GVL.ActVel_RPM_RR - Rr_Speed_rpm;
	//RL_SpeedError := GVL.ActVel_RPM_RL - Rl_Speed_rpm;

ELSE

    RR_Shift_leavel := 1;
    RL_Shift_leavel := 2;
	//RR_SpeedError := Rr_Speed_rpm - GVL.ActVel_RPM_RR;
	//RL_SpeedError := Rl_Speed_rpm - GVL.ActVel_RPM_RL;

END_IF;

//------------------------------------------------------
// RR减速判断
//------------------------------------------------------

IF RR_SpeedError > 5 THEN

    RR_Decelerating := TRUE;

ELSIF RR_SpeedError < 1 THEN

    RR_Decelerating := FALSE;

END_IF;


//------------------------------------------------------
// RL减速判断
//------------------------------------------------------

IF RL_SpeedError > 5 THEN

    RL_Decelerating := TRUE;

ELSIF RL_SpeedError < 1 THEN

    RL_Decelerating := FALSE;

END_IF;

//------------------------------------------------------
// RR P制动
//------------------------------------------------------

IF RR_Decelerating THEN

    RR_BrakeTorque :=
        BrakeKp * RR_SpeedError;

    IF RR_BrakeTorque > BrakeTorqueMax THEN
        RR_BrakeTorque := BrakeTorqueMax;
    END_IF;

    RR_TorqueCmd :=
        -REAL_TO_INT(RR_BrakeTorque * 10);

ELSE

    RR_TorqueCmd := 0;

END_IF;


//------------------------------------------------------
// RL P制动
//------------------------------------------------------

IF RL_Decelerating THEN

    RL_BrakeTorque :=
        BrakeKp * RL_SpeedError;

    IF RL_BrakeTorque > BrakeTorqueMax THEN
        RL_BrakeTorque := BrakeTorqueMax;
    END_IF;

    RL_TorqueCmd :=
        -REAL_TO_INT(RL_BrakeTorque * 10.0);

ELSE

    RL_TorqueCmd := 0;

END_IF;




(*
====================================================================
 8. 急停逻辑
====================================================================
*)
//遥控器急停按键
IF GVL.Emergency_Stop THEN

    BrakeRequest := TRUE;

    Rr_Speed_rpm := 0.0;
    Rl_Speed_rpm := 0.0;

END_IF;

//触边传感器急停

IF GVL.IsCollisionF OR GVL.IsCollisionR THEN

    BrakeRequest := TRUE;

    Rr_Speed_rpm := 0.0;
    Rl_Speed_rpm := 0.0;

END_IF;


(*
====================================================================
 9. 驻车按键
====================================================================
*)
rTrigBtn(CLK := GVL.Remote_Break);

// 按键翻转
IF rTrigBtn.Q THEN
    ParkingState := NOT ParkingState;
END_IF;

// 驻车压力
IF ParkingState THEN

    BrakeRequest := TRUE;

    Rr_Speed_rpm := 0.0;
    Rl_Speed_rpm := 0.0;

END_IF;
(*
=========================================================
统一制动处理
=========================================================
*)

IF BrakeRequest THEN

    PressureValue := 60;

    Enable_Motor := FALSE;

    Rr_Speed_rpm := 0.0;
    Rl_Speed_rpm := 0.0;

ELSE

    PressureValue := 0;

    Enable_Motor := TRUE;

END_IF;

//====================================================================
// 切换驱动模式
//====================================================================
//RR
IF RR_Decelerating THEN
    Motor_Drive_mode_RR := FALSE;      // 扭矩模式
ELSE
    Motor_Drive_mode_RR := TRUE;       // 速度模式
END_IF;

//RL
IF RL_Decelerating THEN
    Motor_Drive_mode_RL := FALSE;
ELSE
    Motor_Drive_mode_RL := TRUE;
END_IF;

(*
====================================================================
 	下发电机控制指令
====================================================================
*)   

fbMotorCmd_RL(
	CanID := 16#10FFE597,
	Gear_Cmd := RL_Shift_leavel,
	DriveMode := Motor_Drive_mode_RL,
	MCU_Enable := Enable_Motor,
	SpeedCmd := LREAL_TO_UINT(Rl_Speed_rpm),
	TorqueCmd := RL_TorqueCmd,
	TxFrame	=> GVL.CAN_Motor_Cmd_RL,
	UdpTxFrame => GCAN212_Send_RL_cmd);
	
fbMotorCmd_RR(
	CanID := 16#10FFE597,
	Gear_Cmd := RR_Shift_leavel,
	DriveMode := Motor_Drive_mode_RR,
	MCU_Enable := Enable_Motor,
	SpeedCmd := LREAL_TO_UINT(Rr_Speed_rpm),
	TorqueCmd := RR_TorqueCmd_test,
	TxFrame	=> GVL.CAN_Motor_Cmd_RR,
	UdpTxFrame => GCAN212_Send_RR_cmd);
(*
====================================================================
 	下发制动指令
====================================================================
*)

VCU_SEB_Req_Data[0] := 6;
VCU_SEB_Req_Data[3] := PressureValue;

(*
====================================================================
 15. 底盘反解车速
====================================================================
*)

fbDepack_MotorStatus1_RL(RxData := GVL.GCAN212_Recive_RL_status1,
						 SpeedFdk => GVL.ActVel_RPM_RL);
fbDepack_MotorStatus1_RR(RxData := GVL.GCAN212_Recive_RR_status1,
						 SpeedFdk => GVL.ActVel_RPM_RR);


fbInvKine(
    ActVel_RL     :=  GVL.ActVel_RPM_RL,
    ActVel_RR     :=  GVL.ActVel_RPM_RR ,
    SteerAngle_FL := fbKine.deltaL,
    SteerAngle_FR := fbKine.deltaR,
    radius        := fbKine.radius
);



(*
====================================================================
 16. 回传遥控器 PDO 数据
====================================================================
*)
IF ReciveCanID = 16#444 THEN
	YkqRxPDO0_data[0] := ReciveCanData[6];

END_IF;


YkqRxPDO0_data[1] :=
    LREAL_TO_BYTE(fbInvKine.VehicleSpeed * 10);

END_FUNCTION_BLOCK

// Device/Application/FB_CAN_MCU_Command
FUNCTION_BLOCK FB_CAN_MCU_Command
VAR_INPUT
	CanID          : UDINT;      // CAN扩展帧ID
	//控制命令
	Gear_Cmd      : BYTE;      // 0=N 1=D 2=R
    DriveMode     : BOOL;      // FALSE=Torque  TRUE=Speed
    MCU_Enable    : BOOL;      // FALSE=Disable TRUE=Enable

    TorqueCmd     : INT;      // Nm，0.1Nm/bit，负值表示制动
    SpeedCmd      : UINT;      // rpm，1rpm/bit
END_VAR
VAR_OUTPUT
	TxFrame : ARRAY[0..7] OF BYTE;
	UdpTxFrame  : ARRAY[0..12] OF BYTE;     // GCAN212 UDP发送数据
END_VAR
VAR
	Torque_Raw: INT;
    Speed_Raw: UINT;
END_VAR

//======================================================
// Byte0：控制位
//======================================================
TxFrame[0] := 16#00;



// Bit0~1：档位
TxFrame[0] := TxFrame[0] OR UINT_TO_BYTE(Gear_Cmd AND 16#03);

// Bit2：驱动模式
IF DriveMode THEN
    TxFrame[0] := TxFrame[0] OR 16#04;
END_IF;

// Bit3：控制器使能
IF MCU_Enable THEN
    TxFrame[0] := TxFrame[0] OR 16#08;
END_IF;

//======================================================
// Byte1~2：TorqueCmd（INT16，小端）
//======================================================
Torque_Raw := REAL_TO_INT(TorqueCmd * 10.0);

TxFrame[1] := UINT_TO_BYTE(INT_TO_UINT(Torque_Raw) AND 16#00FF);
TxFrame[2] := UINT_TO_BYTE(SHR(INT_TO_UINT(Torque_Raw),8));

//======================================================
// Byte3~4：SpeedCmd（UINT16，小端）
//======================================================
Speed_Raw := SpeedCmd;

TxFrame[3] := UINT_TO_BYTE(Speed_Raw AND 16#00FF);
TxFrame[4] := UINT_TO_BYTE(SHR(Speed_Raw,8));

//======================================================
// Byte5~7：Reserve
//======================================================
TxFrame[5] := 16#00;
TxFrame[6] := 16#00;
TxFrame[7] := 16#00;


//======================================================
// GCAN212 UDP封装
//======================================================

// Byte0
// 扩展帧 + 数据帧 + UDP + DLC=8
UdpTxFrame[0] := 16#A8;

//------------------------------------------------------
// CAN ID（大端）
//------------------------------------------------------
UdpTxFrame[1] := UDINT_TO_BYTE(SHR(CanID,24) AND 16#FF);
UdpTxFrame[2] := UDINT_TO_BYTE(SHR(CanID,16) AND 16#FF);
UdpTxFrame[3] := UDINT_TO_BYTE(SHR(CanID,8)  AND 16#FF);
UdpTxFrame[4] := UDINT_TO_BYTE(CanID AND 16#FF);

//------------------------------------------------------
// CAN DATA
//------------------------------------------------------
UdpTxFrame[5]  := TxFrame[0];
UdpTxFrame[6]  := TxFrame[1];
UdpTxFrame[7]  := TxFrame[2];
UdpTxFrame[8]  := TxFrame[3];
UdpTxFrame[9]  := TxFrame[4];
UdpTxFrame[10] := TxFrame[5];
UdpTxFrame[11] := TxFrame[6];
UdpTxFrame[12] := TxFrame[7];

END_FUNCTION_BLOCK

// Device/Application/FB_Depack_MotorStatus1
FUNCTION_BLOCK FB_Depack_MotorStatus1
VAR_INPUT
    RxData : ARRAY[0..7] OF BYTE;
END_VAR

VAR_OUTPUT
    // Byte0
    Gear_State         : BYTE;      // 0=N 1=D 2=R
    DriveMode_State    : BOOL;      // FALSE=Torque TRUE=Speed
    MCU_Enable_State   : BOOL;

    // Byte1~2
    TorqueFdk_Raw      : INT;       // 原始值
    TorqueFdk          : REAL;      // Nm

    // Byte3~4
    SpeedFdk           : INT;       // rpm

    // Byte5
    MotorTemp_Raw      : BYTE;
    MotorTemp          : INT;       // ℃

    // Byte6
    ControlTemp_Raw    : BYTE;
    ControlTemp        : INT;       // ℃

    // Byte7
    ErrorCode          : BYTE;
END_VAR

VAR
    TempWord : WORD;
END_VAR

//==================== Byte0 ====================

Gear_State := RxData[0] AND 16#03;

DriveMode_State :=
    (RxData[0] AND 16#04) <> 0;

MCU_Enable_State :=
    (RxData[0] AND 16#08) <> 0;


//==================== Torque ====================

TempWord :=
    SHL(BYTE_TO_WORD(RxData[2]),8)
    OR BYTE_TO_WORD(RxData[1]);

TorqueFdk_Raw := WORD_TO_INT(TempWord);

TorqueFdk := INT_TO_REAL(TorqueFdk_Raw) * 0.1;


//==================== Speed ====================

TempWord :=
    SHL(BYTE_TO_WORD(RxData[4]),8)
    OR BYTE_TO_WORD(RxData[3]);

SpeedFdk := WORD_TO_INT(TempWord);


//==================== Temperature ====================

MotorTemp_Raw := RxData[5];
MotorTemp := BYTE_TO_INT(RxData[5]) - 40;

ControlTemp_Raw := RxData[6];
ControlTemp := BYTE_TO_INT(RxData[6]) - 40;


//==================== Error ====================

ErrorCode := RxData[7];

END_FUNCTION_BLOCK

// Device/Application/FB_Depack_MotorStatus2
FUNCTION_BLOCK FB_Depack_MotorStatus2
VAR_INPUT
	RxData : ARRAY[0..7] OF BYTE;
END_VAR
VAR_OUTPUT
	// Byte0~1
    Udc_Raw     : UINT;
    Udc         : REAL;      // V 母线电压

    // Byte2~3
    Idc_Raw     : INT;
    Idc         : REAL;      // A 母线电流

    // Byte4~5
    Iphase_Raw  : UINT;
    Iphase      : REAL;      // A  相电流有效值

    // Byte6~7
    LimitWord   : WORD;

    Limit_OverTemp            : BOOL;		//过温限功率
    Limit_MotorCurrent         : BOOL;		//电机电流限功率
    Limit_UnderVoltage         : BOOL;		//欠压限功率
    Limit_BusCurrent           : BOOL;		//母线电流限功率
    Limit_OverSpeed            : BOOL;		//转速超限限功率
    CurrentSensorFault         : BOOL;		//电流传感器异常
    BusCurrentSensorFault      : BOOL;		//母线电流传感器异常
    EncoderFault               : BOOL;		//编码器异常
    OverLoadLimit              : BOOL;		//过载限功率
    OverPowerLimit             : BOOL;		//超功率限制
END_VAR
VAR
	TempWord : WORD;
END_VAR

//==================== Udc ====================

TempWord :=
    SHL(BYTE_TO_WORD(RxData[1]),8)
    OR BYTE_TO_WORD(RxData[0]);

Udc_Raw := WORD_TO_UINT(TempWord);
Udc := UINT_TO_REAL(Udc_Raw) * 0.1;


//==================== Idc ====================

TempWord :=
    SHL(BYTE_TO_WORD(RxData[3]),8)
    OR BYTE_TO_WORD(RxData[2]);

Idc_Raw := WORD_TO_INT(TempWord);
Idc := INT_TO_REAL(Idc_Raw) * 0.1;


//==================== Iphase ====================

TempWord :=
    SHL(BYTE_TO_WORD(RxData[5]),8)
    OR BYTE_TO_WORD(RxData[4]);

Iphase_Raw := WORD_TO_UINT(TempWord);
Iphase := UINT_TO_REAL(Iphase_Raw) * 0.1;


//==================== Limit Flags ====================

LimitWord :=
    SHL(BYTE_TO_WORD(RxData[7]),8)
    OR BYTE_TO_WORD(RxData[6]);

Limit_OverTemp :=
    (LimitWord AND 16#0001) <> 0;

Limit_MotorCurrent :=
    (LimitWord AND 16#0002) <> 0;

Limit_UnderVoltage :=
    (LimitWord AND 16#0004) <> 0;

Limit_BusCurrent :=
    (LimitWord AND 16#0008) <> 0;

Limit_OverSpeed :=
    (LimitWord AND 16#0010) <> 0;

CurrentSensorFault :=
    (LimitWord AND 16#0020) <> 0;

BusCurrentSensorFault :=
    (LimitWord AND 16#0040) <> 0;

EncoderFault :=
    (LimitWord AND 16#0080) <> 0;

OverLoadLimit :=
    (LimitWord AND 16#0100) <> 0;

OverPowerLimit :=
    (LimitWord AND 16#0200) <> 0;

END_FUNCTION_BLOCK

// Device/Application/FB_AckermannKinematics
FUNCTION_BLOCK FB_AckermannKinematics
VAR_INPUT
	v_kmh		:	LREAL;	//前进速度（km/h)，车辆质心
	delta	:	LREAL;	//等效前轮转角（rad）
	Dir_LR 	: BYTE;
END_VAR
VAR_OUTPUT
	deltaL  : LREAL;  // 左前轮转角 (rad)
    deltaR  : LREAL;  // 右前轮转角 (rad)
    wRL_rpm     : LREAL;  // 左后轮角速度 (rpm)
    wRR_rpm     : LREAL;  // 右后轮角速度 (rpm)
	radius   : LREAL;   // 转弯半径
END_VAR

VAR
	v_ms   :	LREAL;	//前进速度m/s
	L   : LREAL := 1.4;   // 轴距 m
    W   : LREAL := 1.150;   // 轮距 m
    rRL : LREAL := 0.25;   // 左后轮半径 m
    rRR : LREAL := 0.25;   // 右后轮半径 m
    eps : LREAL := 1E-6;   // 防止除零
	
	
    psiDot  : LREAL;   // 偏航角速度 rad/s
    vRL     : LREAL;   // 左后轮线速度
    vRR     : LREAL;   // 右后轮线速度
	tmp 	: LREAL;
	
END_VAR



v_ms := v_kmh / 3.6;  // km/h  ->  m/s

IF ABS(delta) < eps THEN
	radius := 1.0E12;  
	psiDot := 0;
	deltaL := 0;
	deltaR := 0;
	vRL := v_ms;
	vRR := v_ms;
ELSE
	radius := ABS((L/2) / TAN(delta));  //根据自行车模型算出车体转弯半径
	psiDot := v_ms / radius;
	
	deltaL := ATAN(L/2/(radius-W/2)); // 双阿克曼，前后轮转角相同，所以只以前轮计算
	deltaR := ATAN(L/2/(radius+W/2));
	
	vRL := psiDot * SQRT( EXPT((radius - W/2),2) + EXPT(L/2,2) ); //车轮的线速度 m/s
	vRR := psiDot * SQRT( EXPT((radius + W/2),2) + EXPT(L/2,2) );
END_IF

IF Dir_LR  = 2 THEN //右转
	tmp := vRL;
	vRL := vRR;
	vRR := tmp;
END_IF

wRL_rpm := vRL / rRL * 60 / (2*3.1415926);  //车轮转速 rpm
wRR_rpm := vRR / rRR * 60 / (2*3.1415926);

END_FUNCTION_BLOCK

// Device/Application/FB_AckermannInverseKinematics
FUNCTION_BLOCK FB_AckermannInverseKinematics
VAR_INPUT
	ActVel_RL    : DINT;   // 左后轮速度反馈 rpm
    ActVel_RR    : DINT;   // 右后轮速度反馈 rpm
    SteerAngle_FL: LREAL;  // 左前轮转角 (rad)
    SteerAngle_FR: LREAL;  // 右前轮转角 (rad)
	radius		 : LREAL;   		//转弯半径
END_VAR
VAR_OUTPUT
	VehicleSpeed : REAL; // 车辆质心速度 (km/h)
	delta		: REAL;  //车轮转向角
    //HeadingAngle : LREAL; // 航向角 (rad)
END_VAR
VAR
	L	:	REAL := 1.4;  //轴距
	v_RL, v_RR   : REAL; // 后轮线速度
    v_rear       : LREAL; // 后轴平均速度
    R_L, R_R     : LREAL; // 由左右前轮计算的转弯半径
    R_avg        : LREAL; // 平均转弯半径
	
	wheelRadius  : LREAL:= 0.25;  // 车轮半径 (m)
    axleLength   : LREAL := 1.4;  // 前后轴距 (m)
    trackWidth   : LREAL := 1.150;  // 前轮轮距 (m)
	eps : LREAL := 1E-6;   // 防止除零
	
	cosL    : REAL;
    cosR    : REAL;
	delta_L     : REAL;   // 左前=左后轮转角 [rad]，正值向左转
    delta_R     : REAL;   // 右前=右后轮转角 [rad]，正值向右转
END_VAR

// ============= 逆运动学计算 =============
IF ActVel_RL < 0 THEN
	ActVel_RL := -ActVel_RL;
END_IF
IF ActVel_RR < 0 THEN
	ActVel_RR := -ActVel_RR;
END_IF
// 1. 单位换算：rpm -> m/s
v_RL := DINT_TO_REAL(ActVel_RL) / 60.0 * 2.0 * 3.14159 * wheelRadius;
v_RR := DINT_TO_REAL(ActVel_RR) / 60.0 * 2.0 * 3.14159 * wheelRadius;

delta_L := ATAN((L/2) / (radius-trackWidth/2));
delta_R := ATAN((L/2) / (radius+trackWidth/2));


// 2. 核心公式：纵向速度 = 左右后轮纵向分速平均
cosL := COS(delta_L);
cosR := COS(delta_R);
// 防止 cos 接近0时数值爆炸（极端蟹行）
IF cosL < 0.05 THEN cosL := 0.05; END_IF;
IF cosR < 0.05 THEN cosR := 0.05; END_IF;

VehicleSpeed := (v_RL * cosL + v_RR * cosR) / 2.0 * 3.6;  //km/h

delta := ATAN((L/2)/radius);

END_FUNCTION_BLOCK

// Device/Application/FB_MoveByFSD
FUNCTION_BLOCK FB_MoveByFSD
VAR_INPUT
	//recvBuf : ARRAY[0..12] OF BYTE;
	//UDP_RecvBuf     : ARRAY[0..12] OF BYTE;  //UDP接收数据
	//			:	BOOL;				//初始化标志 ，没用到
END_VAR
VAR_OUTPUT
	//UDP_SendBuf_RR_Motor_Cmd     : ARRAY[0..12] OF BYTE;		//	UDP发送数据
	//UDP_SendBuf_RL_Motor_Cmd     : ARRAY[0..12] OF BYTE;
END_VAR
VAR
(*
====================================================================
运动学功能块
====================================================================
*)
	
	fbKine			:	FB_AckermannKinematics;
	fbInvKine		:	FB_AckermannInverseKinematics;


	(* 急停释放检测 *)
    xStopState : BOOL;

(*
====================================================================
CAN协议解析
====================================================================
*)
	CAN_SCU1_Recv	:	FB_CAN_SCU_1;	//
	CAN_CCU_Send	:	FB_CAN_CCU;
	CAN_BMS_Send	:	FB_CAN_BMS;
	
(*
====================================================================
CAN接收
====================================================================
*)	
//从智驾层接收到的信号
// 	CANBus_DevRxMsg_0: CANBus_DevRxMsg;
// 	rx_enable	:	BOOL;
// 	rx_DexId	:	UINT;
// 	Rx_FilterMsg	:	CANBus_RxFilter_t;
// 	RxMsg	:	CANBus_FrameMsg_t;
// 	error_ID	:	CANBus_FBErrorType_Enum;
	
(*
====================================================================
车辆目标指令
====================================================================
*)	
	Target_ForwardWheelAngle	:	LREAL;
	Target_ReardWheelAngleMap		:	LREAL;
	Target_ReardWheelAngle		:	LREAL;
	Target_Speed	:	LREAL;

(*
====================================================================
CAN数据缓存
====================================================================
*)
	//给智驾发送的CNA数据
	BMS_Send_Data	:	ARRAY[0..7] OF BYTE;
	CCU_CAN_Data	:	ARRAY[0..7] OF BYTE;
	//检测udp接收超时
	udiNowTime      : UDINT;
    udiLastChangeTime   : UDINT;
	UDP_TimeFrame	:	UINT;
	UDP_TimeFrame_Pre	:	UINT;
	UDP_RX_Timeout	:	BOOL := FALSE;
(*
====================================================================
车轮转向角
====================================================================
*)
	Angle_RL	:	LREAL;
	Angle_RR	:	LREAL;
	Angle_FL	:	LREAL;
	Angle_FR	:	LREAL;
(*
====================================================================
车轮速度
====================================================================
*)
	Speed_RR	:	LREAL;
	Speed_RL	:	LREAL;

(*
====================================================================
整车状态
====================================================================
*)
	Vehicle_Speed	:	REAL;
	Steering_Wheel_Angle	:	REAL;
	radius   : LREAL;   // 转弯半径
	
	Vehicle_ShiftLevel	:	UINT;
	
	//电机状态解包
	fbDepack_MotorStatus1_RR	:	FB_Depack_MotorStatus1;
	fbDepack_MotorStatus2_RR	:	FB_Depack_MotorStatus2;
	fbDepack_MotorStatus1_RL	:	FB_Depack_MotorStatus1;
	fbDepack_MotorStatus2_RL	:	FB_Depack_MotorStatus2;
	
(*
====================================================================
安全状态
====================================================================
*)
   	
	//触边
	
	//刹车
	Break	:	BOOL ;
	//档位
	ShiftLevel	:	UINT;
	

(*
====================================================================
转向机构参数
====================================================================
*)
	//转向
	Ls_mm    : REAL := 100.0;   // 转向节转臂长度 (mm)
    Pitch_mm : REAL := 43.692;  // 转向器线角比 (mm/rev)

    RackTravel_mm : REAL;       // 拉杆位移
    PI            : REAL := 3.1415926;
	Ratio       : REAL;         // 归一化比例 0.0~1.0
    //SteeringDeg : REAL;         // 前轮转向角度（度）
    SteeringRad : REAL;         // 前轮转角（rad）
    SteerAngle_deg : REAL;      // 转向器目标角度（deg）
	Target_ReardWheelAngleAbs: LREAL;
    Dir_LR : BYTE;
(*
====================================================================
下发电机控制指令
====================================================================
*)	
	fbMotorCmd_RR		:	FB_CAN_MCU_Command;
	fbMotorCmd_RL		:	FB_CAN_MCU_Command;
	//车辆行驶档位  0:N  1:D  2:R
	RR_Shift_leavel	:	BYTE;   
	RL_Shift_leavel	:	BYTE;
	//电机驱动方式  1:速度  0:力矩
	Motor_Drive_mode_RR	:	BOOL := 1 ;
	Motor_Drive_mode_RL	:	BOOL := 1 ;
	Eanble_Motor	:	BOOL:=TRUE;
(*
====================================================================
制动系统相关指令
====================================================================
*)
	PressureValue	: BYTE;
	BrakeRequest : BOOL := FALSE;
	
(*
====================================================================
调试变量
====================================================================
*)	
	test : BOOL := TRUE;

	Target_SpeedTest	:	LREAL;
	Target_ReardWheelAngleTest		:	LREAL;
	
END_VAR

(*
====================================================================
 自动驾驶模式主控制逻辑
 功能：
 1. 自动驾驶初始化
 2. CAN 指令解析
 3. 底盘运动学解算
 4. 驱动轮速度控制
 5. 转向执行
 6. 急停 / 防撞 / 制动逻辑
 7. 整车状态回传
====================================================================
*)

(*
====================================================================
 0. CAN数据接收
====================================================================
*)


(*
====================================================================
 3. 自动驾驶 CAN 指令解析
====================================================================
*)
//IF ReciveCanID = 16#121 THEN

    // 解析 SCU 控制报文
    CAN_SCU1_Recv(
        RawFrame                      := GVL.UDP_Re_FSD_Cmd,
        SCU_Brk_En                    => Break,
        SCU_Target_Speed              => Target_Speed,
        SCU_Steering_Wheel_Angle_F    => Target_ReardWheelAngleMap,
		SCU_ShiftLevel_Req			  => ShiftLevel,
		Time_Frame					  => UDP_TimeFrame
    );

//END_IF;
Target_ReardWheelAngle := Target_ReardWheelAngleMap / 4.444;
IF Target_ReardWheelAngle > 20 THEN
	Target_ReardWheelAngle := 20;
ELSIF Target_ReardWheelAngle < -20 THEN
	Target_ReardWheelAngle := -20;
END_IF

//清空刹车需求
BrakeRequest := FALSE;

(*
====================================================================
 4. 底盘运动学正解
 输入：
    Target_Speed             目标车速
    Target_ReardWheelAngle   目标转角
 输出：
    左右轮转速
    左右轮转角
====================================================================
*)
//增加一个转向方向1,2
Target_ReardWheelAngleAbs := ABS(Target_ReardWheelAngle);
IF Target_ReardWheelAngle >=0 THEN
	Dir_LR := 1;
ELSE
	Dir_LR:=2;
END_IF

fbKine(
    v_kmh  := Target_Speed,
    delta  := Target_ReardWheelAngleAbs * PI / 180,
	Dir_LR := Dir_LR,
    deltaL => Angle_RL,
    deltaR => Angle_RR,

    wRL_rpm => Speed_RL,
    wRR_rpm => Speed_RR,

    radius => radius
);


(*
====================================================================
 5. 单 / 双阿克曼模式切换
====================================================================
*)
IF GVL.AckermanModleTransfer THEN

    // 单阿克曼模式
    Angle_FL := 0.0;
    Angle_FR := 0.0;

ELSE

    // 双阿克曼模式
    Angle_FL := Angle_RL;
    Angle_FR := Angle_RR;

END_IF;


(*
====================================================================
 6. 碰撞保护
====================================================================
*)
IF GVL.IsCollisionF OR GVL.IsCollisionR THEN

    BrakeRequest := TRUE;

END_IF;


(*
====================================================================
 7. 制动 / 急停保护
====================================================================
*)
xStopState := Break OR GVL.Emergency_Stop;

IF xStopState THEN

    BrakeRequest := TRUE;

END_IF;


(*
====================================================================
档位判断
0、2:空挡  1:D   2:R
====================================================================
*)

CASE ShiftLevel OF
	0:
		Speed_RR :=0;
		Speed_RL :=0;
		Vehicle_ShiftLevel := 0;
		BrakeRequest := TRUE;
		
	2:
		Speed_RR :=0;
		Speed_RL :=0;
		Vehicle_ShiftLevel:= 2;
		BrakeRequest := TRUE;
		
	1:  //前进

		RR_Shift_leavel := 2;
		RL_Shift_leavel := 1;
		Vehicle_ShiftLevel:=1;
		
		
	3:	//后退
		RR_Shift_leavel := 1;
		RL_Shift_leavel := 2;
		Vehicle_ShiftLevel:= 3;
		
ELSE
	;
END_CASE



(*
====================================================================
指令接收超时停止
====================================================================
*)
udiNowTime := SysTimeGetMs();
IF UDP_TimeFrame <> UDP_TimeFrame_Pre THEN
	UDP_TimeFrame_Pre := UDP_TimeFrame;
	udiLastChangeTime := udiNowTime;
	UDP_RX_Timeout := FALSE;
ELSE
	//判断时间
	IF  (udiNowTime - udiLastChangeTime) >= 1000 THEN
		UDP_RX_Timeout := TRUE;
	ELSE 
		UDP_RX_Timeout := FALSE;
	END_IF
END_IF


IF UDP_RX_Timeout THEN

    BrakeRequest := TRUE;

END_IF;

(*
=========================================================
统一制动处理
=========================================================
*)

IF BrakeRequest THEN

    Speed_RR := 0.0;
    Speed_RL := 0.0;

    PressureValue := 60;

    Eanble_Motor := FALSE;

ELSE

    PressureValue := 0;

    Eanble_Motor := TRUE;

END_IF;

(*
====================================================================
	下发电机控制指令
====================================================================
*)

fbMotorCmd_RR(
	CanID := 16#10FFE597,
	Gear_Cmd := RR_Shift_leavel,
	DriveMode := Motor_Drive_mode_RR,
	MCU_Enable := Eanble_Motor,
	SpeedCmd := LREAL_TO_UINT(Speed_RR),
	TxFrame	=> GVL.CAN_Motor_Cmd_RR,
	UdpTxFrame => GCAN212_Send_RR_cmd);
fbMotorCmd_RL(
	CanID := 16#10FFE597,
	Gear_Cmd := RL_Shift_leavel,
	DriveMode := Motor_Drive_mode_RL,
	MCU_Enable := Eanble_Motor,
	SpeedCmd := LREAL_TO_UINT(Speed_RL),
	TxFrame	=> GVL.CAN_Motor_Cmd_RL,
	UdpTxFrame => GCAN212_Send_RL_cmd);
(*
====================================================================
 	下发制动指令
====================================================================
*)  
VCU_SEB_Req_Data[0] := 6;
VCU_SEB_Req_Data[3] := PressureValue;
	

(*
====================================================================
 11. 转向执行
====================================================================
*)

// 角度 -> 弧度
SteeringRad :=
    Target_ReardWheelAngle * 3.1415926 / 180.0;

// 轮胎转角 -> 齿条位移
RackTravel_mm :=
    Ls_mm * SteeringRad;

// 齿条位移 -> 转向器角度
SteerAngle_deg :=
    (RackTravel_mm / Pitch_mm) * 360.0;

(*
--------------------------------------------------------------------
 前桥转向 CAN 报文
--------------------------------------------------------------------
*)
CAN_SES_Req_F(
    Tgt_StrAngle    := SteerAngle_deg,
	//Tgt_StrAngle    := 0,
    Tgt_StrAngleSpd := 200,
    Veh_Spd         := 50,
    Enable          := 1,

    CanData => CAN_SES_Req_Data_F
);


(*
--------------------------------------------------------------------
 后桥转向 CAN 报文
--------------------------------------------------------------------
*)
CAN_SES_Req_R(
    Tgt_StrAngle    := -SteerAngle_deg,
	//Tgt_StrAngle    := 0,
    Tgt_StrAngleSpd := 200,
    Veh_Spd         := 50,
    Enable          := 1,

    CanData => CAN_SES_Req_Data_R
);


(*
====================================================================
 13. 底盘运动学反解
====================================================================
*)
fbDepack_MotorStatus1_RL(RxData := GVL.GCAN212_Recive_RL_status1);
fbDepack_MotorStatus2_RL(RxData := GVL.GCAN212_Recive_RL_status2);

fbInvKine(
    ActVel_RL     :=  fbDepack_MotorStatus1_RL.SpeedFdk,
    ActVel_RR     :=  fbDepack_MotorStatus1_RR.SpeedFdk ,

    SteerAngle_FL := fbKine.deltaL,
    SteerAngle_FR := fbKine.deltaR,

    radius        := radius,

    VehicleSpeed  => Vehicle_Speed
);


(*
====================================================================
 14. 整车状态 CAN 回传
====================================================================
*)
CAN_CCU_Send(
    CCU_ShiftLevel_Sts        := Vehicle_ShiftLevel,
    CCU_P_Sts                 := GVL.Emergency_Stop OR GVL.Remote_Break OR Break,
    CCU_Ignition_Sts          := 1,
    CCU_Drive_Mode_Shift      := 0,

    Steering_Wheel_Direction  := TRUE,

    CCU_Steering_Wheel_Angle  := fbInvKine.delta,
    CCU_Vehicle_Speed         := fbInvKine.VehicleSpeed,

    CCU_Drive_Mode            := 1,

    Remote_Brake              := GVL.Remote_Break,
    Emergency_Brake           := GVL.Emergency_Stop,
    SCU_Brake_Singal          := Break,

    Left_Turn_Light_Sts       := test,
    Right_Turn_Light_Sts      := test,

    Position_Light_Sts        := test,
    LowBeam_Sts               := test,

    TxFrame => CCU_CAN_Data
);


(*
====================================================================
 15. BMS 状态转发
====================================================================
*)
IF ReciveCanID = 16#444 THEN

    CAN_BMS_Send(
		RxData := ReciveCanData,
        TxData => BMS_Send_Data
    );
	YkqRxPDO0_data[0] := ReciveCanData[6];
END_IF;
(*
====================================================================
 遥控器显示速度及电量
====================================================================
*)
YkqRxPDO0_data[1] :=
    LREAL_TO_BYTE(fbInvKine.VehicleSpeed * 10);

END_FUNCTION_BLOCK

// Device/Application/test
FUNCTION_BLOCK test
VAR_INPUT
END_VAR
VAR_OUTPUT
END_VAR
VAR
	udp : FB_UDP;
	recvBuf     : ARRAY[0..12] OF BYTE;
	sendBuf     : ARRAY[0..12] OF BYTE := [0,1,2,0,0,0,0,0,0,0,0,0];
	
END_VAR



//udp(sendBuf := sendBuf, recvBuf=>recvBuf);

END_FUNCTION_BLOCK

// Device/Application/FB_CAN_SCU_1
FUNCTION_BLOCK FB_CAN_SCU_1
VAR_INPUT
	RawFrame : ARRAY[0..12] OF BYTE;   // 13字节原始数据
	
END_VAR
VAR_OUTPUT
	SCU_ShiftLevel_Req	:	UINT;; //底盘档位状态
	SCU_Drive_Mode_Req	:	UINT;; //底盘驾驶模式状态
	SCU_Steering_Wheel_Angle_F	:	SINT; //前转向角度控制
	SCU_Steering_Wheel_Angle_R	:	SINT; //后转向角度控制
	SCU_Target_Speed	:	REAL; //速度控制
	SCU_Brk_En	:	BOOL; //刹车信号控制
	GW_Left_Turn_Light_Req	:	UINT; //左转向灯控制
	GW_Right_Turn_Light_Req	:	UINT; //右转向灯控制
	GW_Position_Light_Req	:	UINT; //刹车灯控制
	GW_LowBeam_Req	:	UINT; //近光灯控制
// 	angular_speed_flag	:	INT; //调节转向速度，只部分车型适用
// 	SCU_Brake_Force_Flag	:	BOOL; //调节EMB强度，只针对有EMB的车型
	Time_Frame	:	UINT;	//检测是否超时使用
	
END_VAR
VAR
	// 把13字节里真正的8字节CAN数据取出来（第6~13字节，即索引5~12）
    Data : ARRAY[0..7] OF BYTE;
    
    // 64位无符号整数，用于位字段提取（Intel = Little-Endian）
    Raw64 : ULINT;
    
    i : INT;
END_VAR


//============================================================
// 1. 提取真实的8字节CAN数据（跳过前5字节的长度+ID）
//============================================================
FOR i := 0 TO 7 DO
    //Data[i] := RawFrame[5 + i];
	Data[i] := GVl.UDP_Re_FSD_Cmd[5+i];
END_FOR;

Time_Frame := Data[7];

//============================================================
// 2. Little-Endian 拼成 64bit 整数（最方便做位操作）
//============================================================
Raw64 :=   (SHL(BYTE_TO_ULINT(Data[7]),56))
         OR (SHL(BYTE_TO_ULINT(Data[6]),48))
         OR (SHL(BYTE_TO_ULINT(Data[5]),40))
         OR (SHL(BYTE_TO_ULINT(Data[4]),32))
         OR (SHL(BYTE_TO_ULINT(Data[3]),24))
         OR (SHL(BYTE_TO_ULINT(Data[2]),16))
         OR (SHL(BYTE_TO_ULINT(Data[1]),8))
         OR  BYTE_TO_ULINT(Data[0]);

//============================================================
// 3. 按协议逐个提取信号（全部是 Intel/Little-Endian）
//============================================================

// Startbit 0, Len 2
SCU_ShiftLevel_Req := ULINT_TO_UINT(SHR(Raw64, 0) AND 16#03);

// Startbit 6, Len 2
SCU_Drive_Mode_Req := ULINT_TO_UINT(SHR(Raw64, 6) AND 16#03);

// Startbit 8, Len 8  → Byte1 的高8位
SCU_Steering_Wheel_Angle_F := ULINT_TO_SINT(SHR(Raw64, 8) AND 16#FF);

// Startbit 16, Len 8 → Byte2
SCU_Steering_Wheel_Angle_R := ULINT_TO_SINT(SHR(Raw64,16) AND 16#FF);

// Startbit 24, Len 9  → 跨Byte3[0..7] + Byte4[0]
SCU_Target_Speed := ULINT_TO_REAL(SHR(Raw64,24) AND 16#1FF) * 0.1;

// Startbit 33, Len 1  → Byte4 的 bit1
SCU_Brk_En := (SHR(Raw64,33) AND 16#01) = 16#01;

// Startbit 40, Len 2 → Byte5 bit0~1
GW_Left_Turn_Light_Req  := ULINT_TO_UINT(SHR(Raw64,40) AND 16#03);

// Startbit 42, Len 2 → Byte5 bit2~3
GW_Right_Turn_Light_Req := ULINT_TO_UINT(SHR(Raw64,42) AND 16#03);

// Startbit 46, Len 2 → Byte5 bit6~7
GW_Position_Light_Req   := ULINT_TO_UINT(SHR(Raw64,46) AND 16#03);

// Startbit 48, Len 2 → Byte6 bit0~1
GW_LowBeam_Req          := ULINT_TO_UINT(SHR(Raw64,48) AND 16#03);

// // Startbit 60, Len 1（有符号） → Byte7 bit4
// angular_speed_flag := IF (SHR(Raw64,60) AND 16#01)=1 THEN 1 ELSE 0; // 实际协议里是Signed，但只有0/1
// 
// // Startbit 60, Len 1（无符号） → 同样位置，另一个信号（两个信号重叠bit）
// SCU_Brake_Force_Flag := (SHR(Raw64,60) AND 16#01) = 16#01;

END_FUNCTION_BLOCK

// Device/Application/FB_CAN_CCU
FUNCTION_BLOCK FB_CAN_CCU
VAR_INPUT
	CCU_ShiftLevel_Sts         : UINT;   // 0~3   档位状态
    CCU_P_Sts                  : BOOL;   // 刹车踏板状态
    CCU_Ignition_Sts           : UINT;   // 0~3   点火状态
    CCU_Drive_Mode_Shift       : BOOL;   // 驾驶模式切换按钮
    Steering_Wheel_Direction   : BOOL;   // 前轮转向方向：TRUE=左转，FALSE=右转
    CCU_Steering_Wheel_Angle   : REAL;   // 实际角度 ° → 发送时×10（协议0.1°/LSB，120→12.0°或27°看标定）
    CCU_Vehicle_Speed          : REAL;   // km/h → 发送时×10（0.1km/h 精度）
    CCU_Drive_Mode             : UINT;   // 0~3   当前驾驶模式
    Remote_Brake               : BOOL;   // 遥控器刹车
    Emergency_Brake            : BOOL;   // 紧急制动
    SCU_Brake_Singal           : BOOL;   // 自动驾驶刹车请求
    Left_Turn_Light_Sts        : BOOL;   // 左转灯实际状态
    Right_Turn_Light_Sts       : BOOL;   // 右转灯实际状态
    Position_Light_Sts         : BOOL;   // 刹车灯状态
    LowBeam_Sts                : BOOL;   // 近光灯状态
END_VAR
VAR_OUTPUT
	TxFrame : ARRAY[0..7] OF BYTE;   // 只有数据
END_VAR
VAR
	Raw64      : ULINT := 0;
	Raw64_CAN      : ULINT := 0;
    angle_raw  : UINT;
    speed_raw  : UINT;
	
	i : INT;
    
	nibble : ULINT;
    
END_VAR

//======================================================
// 1. 按 Intel (Little-Endian) 顺序打包所有信号到 64bit
//======================================================
Raw64 := 0;  // 先清零

// bit 0~1: CCU_ShiftLevel_Sts (2 bits)
Raw64 := Raw64 OR SHL(UINT_TO_ULINT(CCU_ShiftLevel_Sts AND 16#03), 0);

// bit 2: CCU_P_Sts
IF CCU_P_Sts THEN
    Raw64 := Raw64 OR SHL(16#1, 2);
END_IF;

// bit 3~4: CCU_Ignition_Sts (2 bits)
Raw64 := Raw64 OR SHL(UINT_TO_ULINT(CCU_Ignition_Sts AND 16#03), 3);

// bit 5: CCU_Drive_Mode_Shift
IF CCU_Drive_Mode_Shift THEN
    Raw64 := Raw64 OR SHL(16#1, 5);
END_IF;

// bit 7: Steering_Wheel_Direction (左1 右0)
IF Steering_Wheel_Direction THEN
    Raw64 := Raw64 OR SHL(16#1, 7);
END_IF;

// bit 8~19: CCU_Steering_Wheel_Angle (12 bits, 0.1°/LSB)
angle_raw := REAL_TO_UINT(CCU_Steering_Wheel_Angle * 10.0);
Raw64 := Raw64 OR SHL(UINT_TO_ULINT(angle_raw AND 16#0FFF), 8);

// bit 20~28: CCU_Vehicle_Speed (9 bits, 0.1 km/h/LSB)
speed_raw := REAL_TO_UINT(CCU_Vehicle_Speed * 10.0);  // 关键：×10
Raw64 := Raw64 OR SHL(UINT_TO_ULINT(speed_raw AND 16#1FF), 20);

// bit 29~31: CCU_Drive_Mode (3 bits)
Raw64 := Raw64 OR SHL(UINT_TO_ULINT(CCU_Drive_Mode AND 16#07), 29);

// bit 32: Remote_Brake
IF Remote_Brake THEN
    Raw64 := Raw64 OR SHL(16#1, 32);
END_IF;

// bit 33: Emergency_Brake
IF Emergency_Brake THEN
    Raw64 := Raw64 OR SHL(16#1, 33);
END_IF;

// bit 34: SCU_Brake_Singal
IF SCU_Brake_Singal THEN
    Raw64 := Raw64 OR SHL(16#1, 34);
END_IF;

// bit 56: Left_Turn_Light_Sts
IF Left_Turn_Light_Sts THEN
    Raw64 := Raw64 OR SHL(16#1, 56);
END_IF;

// bit 57: Right_Turn_Light_Sts
IF Right_Turn_Light_Sts THEN
    Raw64 := Raw64 OR SHL(16#1, 57);
END_IF;

// bit 59: Position_Light_Sts (刹车灯)
IF Position_Light_Sts THEN
    Raw64 := Raw64 OR SHL(16#1, 59);
END_IF;

// bit 60: LowBeam_Sts
IF LowBeam_Sts THEN
    Raw64 := Raw64 OR SHL(16#1, 60);
END_IF;

//======================================================
// 2. 直接拆出 8 字节数据区（Intel 顺序已经是低字节在前）
//======================================================
TxFrame[0]  := ULINT_TO_BYTE(Raw64);           // Data0
TxFrame[1]  := ULINT_TO_BYTE(SHR(Raw64, 8));    // Data1
TxFrame[2]  := ULINT_TO_BYTE(SHR(Raw64, 16));   // Data2
TxFrame[3]  := ULINT_TO_BYTE(SHR(Raw64, 24));   // Data3
TxFrame[4]  := ULINT_TO_BYTE(SHR(Raw64, 32));   // Data4
TxFrame[5] := ULINT_TO_BYTE(SHR(Raw64, 40));   // Data5
TxFrame[6] := ULINT_TO_BYTE(SHR(Raw64, 48));   // Data6
TxFrame[7] := ULINT_TO_BYTE(SHR(Raw64, 56));   // Data7

//======================================================
// 3. 填充前5字节：DLC + CAN ID 0x51 (Standard Frame)
//    常见格式：Big-Endian ID，标准帧通常低字节有效
//======================================================
// TxFrame[0] := 16#08;         // DLC = 8
// 
// TxFrame[1] := 0;             // ID 高字节
// TxFrame[2] := 0;             
// TxFrame[3] := 0;             
// TxFrame[4] := 16#51;          // ID = 0x51，低字节放这里（常见做法）

END_FUNCTION_BLOCK

// Device/Application/FB_CAN_BMS
FUNCTION_BLOCK FB_CAN_BMS
VAR_INPUT
    RxData : ARRAY[0..7] OF BYTE;
END_VAR

VAR_OUTPUT
    TxData : ARRAY[0..7] OF BYTE;   // 仅仅返回CAN数据
END_VAR

VAR
    (* 原始值 *)
    VoltageRaw : UINT;
    CurrentRaw : INT;

    (* 实际值 *)
    VoltageReal : REAL;
    CurrentReal : REAL;

    (* 重新编码后的值 *)
    VoltageSend : UINT;
    CurrentSend : INT;
END_VAR

(* ============================= *)
(* 1. 解析接收到的CAN数据 *)
(* ============================= *)

(* 电压：低字节在前，高字节在后 *)
VoltageRaw := BYTE_TO_UINT(RxData[0]) OR SHL(BYTE_TO_UINT(RxData[1]), 8);

(* 电流：低字节在前，高字节在后 *)
CurrentRaw := BYTE_TO_INT(RxData[2]) OR SHL(BYTE_TO_INT(RxData[3]), 8);


(* ============================= *)
(* 2. 转换为实际物理量 *)
(* ============================= *)

(* 电压：0~4000 -> 0~400V *)
VoltageReal := UINT_TO_REAL(VoltageRaw) * 0.1;

(* 电流：0~1000 -> -500A~500A *)
CurrentReal := INT_TO_REAL(CurrentRaw) - 500.0;


(* ============================= *)
(* 3. 再重新编码 *)
(* ============================= *)


VoltageSend := REAL_TO_UINT(VoltageReal );
CurrentSend := REAL_TO_INT(CurrentReal );


(* ============================= *)
(* 4. 打包成CAN发送数据 *)
(* ============================= *)

(* 电压 *)
TxData[0] := UINT_TO_BYTE(VoltageSend AND 16#00FF);
TxData[1] := UINT_TO_BYTE(SHR(VoltageSend, 8));

(* 电流 *)
TxData[2] := INT_TO_BYTE(CurrentSend AND 16#00FF);
TxData[3] := INT_TO_BYTE(SHR(CurrentSend, 8));

(* 其余字节清零 *)
TxData[4] := RxData[6];
TxData[5] := 0;
TxData[6] := 0;
TxData[7] := 0;

END_FUNCTION_BLOCK

// Device/Application/FB_MoveControlByTorque_Yaokong
FUNCTION_BLOCK FB_MoveControlByTorque_Yaokong
//====================================================================
// 工业级双Ackermann轮毂电机底盘运动控制器 - 遥控器模式
// 版本：V2.5 (按通讯协议 + 速度斜坡 + 移除所有死区)
// 说明：遥控器及电机反馈精确，无需死区处理
//====================================================================

VAR_INPUT
END_VAR

VAR_OUTPUT
END_VAR

//====================================================================
// 遥控器输入
//====================================================================
VAR
    RemoteDriveRaw     : BYTE;
    RemoteSteerRaw     : BYTE;
    DriveCenter        : INT := 16#7F;
    DriveOffset        : INT;
    DriveRatio         : LREAL;
    SteeringRatio      : REAL;
    Dir_LR             : BYTE;
END_VAR

//====================================================================
// 车辆运动控制
//====================================================================
VAR
    TargetSpeedMax_kmh : LREAL;
    TargetSpeed_kmh    : LREAL;      // 遥控器原始目标速度
    SpeedReference     : LREAL := 0.0; // 斜坡后的参考速度
    Rr_Target_rpm      : LREAL;
    Rl_Target_rpm      : LREAL;
    Rr_Actual_rpm      : LREAL;
    Rl_Actual_rpm      : LREAL;
    Rr_SpeedError      : LREAL;
    Rl_SpeedError      : LREAL;
    Enable_Motor       : BOOL := TRUE;
    RR_Shift_leavel    : BYTE;
    RL_Shift_leavel    : BYTE;
END_VAR

//====================================================================
// 转向机构参数
//====================================================================
VAR
    Ls_mm         : REAL := 100.0;
    Pitch_mm      : REAL := 43.692;
    RackTravel_mm : REAL;
    SteerAngle_deg: REAL;
    PI_const      : REAL := 3.1415926;
    SteeringDeg   : REAL;
    SteeringRad   : REAL;
END_VAR

//====================================================================
// 运动学
//====================================================================
VAR
    fbKine   : FB_AckermannKinematics;
    fbInvKine: FB_AckermannInverseKinematics;
END_VAR

//====================================================================
// 电机控制
//====================================================================
VAR
    fbMotorCmd_RR : FB_CAN_MCU_Command;
    fbMotorCmd_RL : FB_CAN_MCU_Command;
END_VAR

//====================================================================
// PI + 前馈控制器
//====================================================================
VAR
    Kp             : LREAL := 3;
    Ki             : LREAL := 0;
    Integral_RR    : LREAL := 0.0;
    Integral_RL    : LREAL := 0.0;
    IntegralLimit  : LREAL := 70.0;
    FeedforwardGain: LREAL := 0.85;
    FF_Torque_RR   : LREAL;
    FF_Torque_RL   : LREAL;
    TotalTorque_RR : LREAL;
    TotalTorque_RL : LREAL;
    TorqueCmd_RR   : INT;
    TorqueCmd_RL   : INT;
    MaxTorque      : LREAL := 130.0;
    MinTorque      : LREAL := -130.0;
END_VAR

//====================================================================
// 速度斜坡参数（适配4ms周期）
//====================================================================
VAR
    RampUpRate     : LREAL := 5.0;    // km/h/s   可根据实际车辆微调
    RampDownRate   : LREAL := 15.0;    // km/h/s
    CycleTimeMs    : LREAL := 4.0;     // PLC实际任务周期
    d_t            : LREAL;
END_VAR

//====================================================================
// 制动与安全
//====================================================================
VAR
    BrakeRequest   : BOOL := FALSE;
    PressureValue  : BYTE := 0;
    rTrigBtn       : R_TRIG;
    ParkingState   : BOOL := FALSE;
END_VAR

//====================================================================
// 电机状态
//====================================================================
VAR
    fbDepack_MotorStatus1_RR : FB_Depack_MotorStatus1;
    fbDepack_MotorStatus1_RL : FB_Depack_MotorStatus1;
	IsReversingAndDecelerating : BOOL := FALSE;   // 正在后退减速过程
END_VAR

(*
====================================================================
 主控制逻辑
====================================================================
*)


(*
1. 遥控器解析 + 目标速度生成（已移除死区）
*)
TargetSpeedMax_kmh := BYTE_TO_LREAL(YkqTxPDO1_data[0]) / 10.0;
RemoteDriveRaw     := YkqTxPDO1_data[1];
RemoteSteerRaw     := YkqTxPDO1_data[2];

DriveOffset := BYTE_TO_INT(RemoteDriveRaw) - DriveCenter;
DriveRatio  := INT_TO_LREAL(DriveOffset) / 127.0;   // 直接线性映射，无死区

IF DriveRatio > 1.0 THEN DriveRatio := 1.0; END_IF;
IF DriveRatio < -1.0 THEN DriveRatio := -1.0; END_IF;

TargetSpeed_kmh := TargetSpeedMax_kmh * DriveRatio;  // 正值前进，负值后退

(*
2. 转向角计算
*)
IF RemoteSteerRaw < 127 THEN 
    Dir_LR := 1; 
ELSE 
    Dir_LR := 2; 
END_IF;
SteeringRatio := BYTE_TO_REAL(RemoteSteerRaw) / 255.0;
SteeringDeg   := -20.0 + (SteeringRatio * 40.0);
SteeringRad   := SteeringDeg * PI_const / 180.0;

(*
3. 转向机构 CAN 下发
*)
RackTravel_mm := Ls_mm * SteeringRad;
SteerAngle_deg := (RackTravel_mm / Pitch_mm) * 360.0;

CAN_SES_Req_F(Tgt_StrAngle := SteerAngle_deg, Tgt_StrAngleSpd := 200, Veh_Spd := 50, Enable := 1);
CAN_SES_Req_Data_F := CAN_SES_Req_F.CanData;

CAN_SES_Req_R(Tgt_StrAngle := -SteerAngle_deg, Tgt_StrAngleSpd := 200, Veh_Spd := 50, Enable := 1);
CAN_SES_Req_Data_R := CAN_SES_Req_R.CanData;

(*
4. 速度斜坡生成 (速度曲线)
*)
d_t := CycleTimeMs / 1000.0;

IF TargetSpeed_kmh > SpeedReference THEN
    SpeedReference := SpeedReference + RampUpRate * d_t;
    IF SpeedReference > TargetSpeed_kmh THEN SpeedReference := TargetSpeed_kmh; END_IF;
ELSE
    SpeedReference := SpeedReference - RampDownRate * d_t;
    IF SpeedReference < TargetSpeed_kmh THEN SpeedReference := TargetSpeed_kmh; END_IF;
END_IF;

(*
5. 运动学正解
*)
fbKine(v_kmh := SpeedReference, delta := ABS(SteeringRad), Dir_LR := Dir_LR);
Rr_Target_rpm := fbKine.wRR_rpm;
Rl_Target_rpm := fbKine.wRL_rpm;

(*
6. 读取实际转速
*)
fbDepack_MotorStatus1_RR(RxData := GVL.GCAN212_Recive_RR_status1);
fbDepack_MotorStatus1_RL(RxData := GVL.GCAN212_Recive_RL_status1);

Rr_Actual_rpm := INT_TO_LREAL(fbDepack_MotorStatus1_RR.SpeedFdk);
Rl_Actual_rpm := INT_TO_LREAL(fbDepack_MotorStatus1_RL.SpeedFdk);

//******判断是否是倒车减速******
IsReversingAndDecelerating := FALSE;
// 判断正在后退且处于减速过程
IF (SpeedReference <= 0 ) AND   // 曾经/当前在后退
   (Rr_Actual_rpm < 0) AND                               // 实际还在明显后退
   (Rr_Target_rpm> Rr_Actual_rpm) THEN                 // 目标速度 >= 当前参考速度（向0或停止靠近）
   
    IsReversingAndDecelerating := TRUE;
END_IF;

(*
7. 误差计算 + 前馈 + PI 控制
*)
Rr_SpeedError := Rr_Target_rpm - Rr_Actual_rpm;
Rl_SpeedError := Rl_Target_rpm - Rl_Actual_rpm;

FF_Torque_RR := Rr_Target_rpm * FeedforwardGain * 0.012;
FF_Torque_RL := Rl_Target_rpm * FeedforwardGain * 0.012;

Integral_RR := Integral_RR + Rr_SpeedError * Ki;
Integral_RL := Integral_RL + Rl_SpeedError * Ki;
Integral_RR := LIMIT(-IntegralLimit, Integral_RR, IntegralLimit);
Integral_RL := LIMIT(-IntegralLimit, Integral_RL, IntegralLimit);

TotalTorque_RR := FF_Torque_RR + Kp * Rr_SpeedError + Integral_RR;
TotalTorque_RL := FF_Torque_RL + Kp * Rl_SpeedError + Integral_RL;

(*
8. 档位处理 + 协议要求的扭矩符号修正
*)
IF DriveRatio > 0.0 THEN        // 前进
    RR_Shift_leavel := 2;
    RL_Shift_leavel := 1;
ELSIF DriveRatio < 0.0 THEN     // 后退
    RR_Shift_leavel := 1;
    RL_Shift_leavel := 2;
ELSIF DriveRatio = 0.0 THEN
    Integral_RR := 0;
    Integral_RL := 0;
END_IF;

// 只在「明显驱动意图」且「速度误差方向与驱动方向一致」时才强制正向力矩
// 否则让PI自然输出负力矩进行减速
IF (ABS(DriveRatio) > 0.05) AND (NOT BrakeRequest) THEN
    IF (DriveRatio > 0.0 AND Rr_SpeedError > 0.0) OR (DriveRatio < 0.0 AND Rr_SpeedError < 0.0) THEN
        TotalTorque_RR := ABS(TotalTorque_RR);
        TotalTorque_RL := ABS(TotalTorque_RL);
    END_IF;
END_IF;
//倒车减速给负值力矩
IF IsReversingAndDecelerating THEN
	TotalTorque_RR := -ABS(TotalTorque_RR);
    TotalTorque_RL := -ABS(TotalTorque_RL);
END_IF

(*
9. 安全保护
*)
BrakeRequest := FALSE;
IF GVL.Emergency_Stop OR GVL.IsCollisionF OR GVL.IsCollisionR THEN
    BrakeRequest := TRUE;
    Integral_RR := 0.0;
    Integral_RL := 0.0;
END_IF;

rTrigBtn(CLK := GVL.Remote_Break);
IF rTrigBtn.Q THEN ParkingState := NOT ParkingState; END_IF;

IF ParkingState THEN
    BrakeRequest := TRUE;
    Integral_RR := 0.0;
    Integral_RL := 0.0;
END_IF;

(*
10. 统一制动处理 + 最终限幅
*)
IF BrakeRequest THEN
    PressureValue := 60;
    Enable_Motor := FALSE;
    TorqueCmd_RR := 0;
    TorqueCmd_RL := 0;
    Integral_RR := 0.0;
    Integral_RL := 0.0;
    SpeedReference := 0.0;
ELSE
    PressureValue := 0;
    Enable_Motor := TRUE;
    
    TotalTorque_RR := LIMIT(MinTorque, TotalTorque_RR, MaxTorque);
    TotalTorque_RL := LIMIT(MinTorque, TotalTorque_RL, MaxTorque);
    

	   TorqueCmd_RR := REAL_TO_INT(TotalTorque_RR );
 	   TorqueCmd_RL := REAL_TO_INT(TotalTorque_RL );
END_IF;

(*
11. 下发电机指令（力矩模式）
*)
fbMotorCmd_RR(
    CanID := 16#10FFE597,
    Gear_Cmd := RR_Shift_leavel,
    DriveMode := FALSE,
    MCU_Enable := Enable_Motor,
    TorqueCmd := TorqueCmd_RR,
    TxFrame => GVL.CAN_Motor_Cmd_RR,
    UdpTxFrame => GVL.GCAN212_Send_RR_cmd
);

fbMotorCmd_RL(
    CanID := 16#10FFE597,
    Gear_Cmd := RL_Shift_leavel,
    DriveMode := FALSE,
    MCU_Enable := Enable_Motor,
    TorqueCmd := TorqueCmd_RL,
    TxFrame => GVL.CAN_Motor_Cmd_RL,
    UdpTxFrame => GVL.GCAN212_Send_RL_cmd
);

(*
12. 制动指令
*)
VCU_SEB_Req_Data[0] := 6;
VCU_SEB_Req_Data[3] := PressureValue;

(*
13. 车速反解与显示
*)
fbInvKine(
    ActVel_RL := fbDepack_MotorStatus1_RL.SpeedFdk,
    ActVel_RR := fbDepack_MotorStatus1_RR.SpeedFdk,
    SteerAngle_FL := fbKine.deltaL,
    SteerAngle_FR := fbKine.deltaR,
    radius := fbKine.radius
);

IF ReciveCanID = 16#444 THEN
    YkqRxPDO0_data[0] := ReciveCanData[6];
END_IF;
YkqRxPDO0_data[1] := LREAL_TO_BYTE(fbInvKine.VehicleSpeed * 10);

END_FUNCTION_BLOCK

// Device/Application/FB_MoveControlByTorque_FSD
FUNCTION_BLOCK FB_MoveControlByTorque_FSD
//====================================================================
// 工业级双Ackermann轮毂电机底盘运动控制器 - 智驾模式
// 版本：V2.1 (结构化优化版)
// 输入来源：智驾层 UDP/CAN 指令
//====================================================================

VAR_INPUT
END_VAR

VAR_OUTPUT
END_VAR
 //反馈给智驾的信息
VAR
	CAN_BMS_Send	:	FB_CAN_BMS;
	CAN_CCU_Send	:	FB_CAN_CCU;
	CCU_CAN_Data	:	ARRAY[0..7] OF BYTE;  //整车状态
	BMS_Send_Data	:	ARRAY[0..7] OF BYTE;
	
END_VAR
//====================================================================
// 智驾指令解析
//====================================================================
VAR
    CAN_SCU1_Recv     : FB_CAN_SCU_1;
    
    Target_Speed      : LREAL;
    Target_ReardWheelAngleMap : LREAL;
    Target_ReardWheelAngle : LREAL;
    ShiftLevel        : UINT := 1;
    Break             : BOOL;
    UDP_TimeFrame     : UINT;
    UDP_TimeFrame_Pre : UINT;
	IsReversingAndDecelerating: BOOL;
END_VAR

//====================================================================
// 速度指令与斜坡
//====================================================================
VAR
    TargetSpeed_kmh    : LREAL;
    SpeedReference     : LREAL;
    
    RampUpRate         : LREAL := 5.0;     // km/h/s
    RampDownRate       : LREAL := 15.0;    // km/h/s
    
END_VAR

//====================================================================
// 转向控制
//====================================================================
VAR
    Ls_mm              : REAL := 100.0;
    Pitch_mm           : REAL := 43.692;
    RackTravel_mm      : REAL;
    SteerAngle_deg     : REAL;
    PI_const           : REAL := 3.1415926;
    SteeringRad        : REAL;
    Target_ReardWheelAngleAbs : LREAL;
    Dir_LR             : BYTE;
END_VAR

//====================================================================
// 运动学
//====================================================================
VAR
    fbKine             : FB_AckermannKinematics;
    fbInvKine          : FB_AckermannInverseKinematics;
END_VAR

//====================================================================
// 电机反馈与状态
//====================================================================
VAR
    Rr_Target_rpm      : LREAL;
    Rl_Target_rpm      : LREAL;
    Rr_Actual_rpm      : LREAL;
    Rl_Actual_rpm      : LREAL;
    Rr_SpeedError      : LREAL;
    Rl_SpeedError      : LREAL;
    
    fbDepack_MotorStatus1_RR : FB_Depack_MotorStatus1;
    fbDepack_MotorStatus1_RL : FB_Depack_MotorStatus1;
END_VAR

//====================================================================
// PI + 前馈 控制器
//====================================================================
VAR
    Kp                 : LREAL := 4;
    Ki                 : LREAL := 0;
    Integral_RR        : LREAL := 0.0;
    Integral_RL        : LREAL := 0.0;
    IntegralLimit      : LREAL := 65.0;
    
    FeedforwardGain    : LREAL := 0.72;
    FF_Torque_RR       : LREAL;
    FF_Torque_RL       : LREAL;
    
    TotalTorque_RR     : LREAL;
    TotalTorque_RL     : LREAL;
    TorqueCmd_RR       : INT;
    TorqueCmd_RL       : INT;
    
    MaxTorque          : LREAL := 130.0;
    MinTorque          : LREAL := -130.0;
END_VAR

//====================================================================
// 停车与零速逻辑
//====================================================================
VAR
    BrakeRequest       : BOOL := FALSE;
    PressureValue      : BYTE := 0;
    Enable_Motor       : BOOL := TRUE;
    
    RR_Shift_leavel    : BYTE;
    RL_Shift_leavel    : BYTE;
    
    // 超时检测
    udiNowTime         : UDINT;
    udiLastChangeTime  : UDINT;
    UDP_RX_Timeout     : BOOL := FALSE;
END_VAR

//====================================================================
// 安全
//====================================================================
VAR
    Vehicle_ShiftLevel : UINT;
END_VAR

//====================================================================
// 电机控制
//====================================================================
VAR
    fbMotorCmd_RR      : FB_CAN_MCU_Command;
    fbMotorCmd_RL      : FB_CAN_MCU_Command;
END_VAR

//====================================================================
// 循环时间
//====================================================================
VAR
    CycleTimeMs        : LREAL := 4.0;
    d_t                 : LREAL;
END_VAR

//====================================================================
// 调试变量
//====================================================================
VAR
    Target_Speed_test : LREAL;
	Target_ReardWheelAngle_test : LREAL;
END_VAR

(*
====================================================================
 主控制循环 - 智驾模式
====================================================================
*)

(*
====================================================
1. 智驾指令解析 (CAN_SCU1)
====================================================
*)
CAN_SCU1_Recv(
    //RawFrame                      := GVL.UDP_Re_FSD_Cmd,
    SCU_Brk_En                    => Break,
    SCU_Target_Speed              => Target_Speed,
    SCU_Steering_Wheel_Angle_F    => Target_ReardWheelAngleMap,
    SCU_ShiftLevel_Req            => ShiftLevel,
    Time_Frame                    => UDP_TimeFrame
);
IF Target_Speed > 5 THEN
	Target_Speed := 5;
END_IF

Target_ReardWheelAngle := Target_ReardWheelAngleMap / 4.444;
IF Target_ReardWheelAngle > 20 THEN
    Target_ReardWheelAngle := 20;
ELSIF Target_ReardWheelAngle < -20 THEN
    Target_ReardWheelAngle := -20;
END_IF;
(*
====================================================
10. 档位判断
====================================================
*)
//测试
//TargetSpeed_kmh := Target_Speed_test;
//ShiftLevel := 1;
CASE ShiftLevel OF
    1:  // 前进
		TargetSpeed_kmh := Target_Speed;
        RR_Shift_leavel := 2;
        RL_Shift_leavel := 1;
        Vehicle_ShiftLevel := 1;
    3:  // 后退
		TargetSpeed_kmh := -Target_Speed;
        RR_Shift_leavel := 1;
        RL_Shift_leavel := 2;
        Vehicle_ShiftLevel := 3;
ELSE
    ;
END_CASE;



(*
====================================================
2. 指令超时检测
====================================================
*)
udiNowTime := SysTimeGetMs();
IF UDP_TimeFrame <> UDP_TimeFrame_Pre THEN
    UDP_TimeFrame_Pre := UDP_TimeFrame;
    udiLastChangeTime := udiNowTime;
    UDP_RX_Timeout := FALSE;
ELSE
    IF (udiNowTime - udiLastChangeTime) >= 1000 THEN
        UDP_RX_Timeout := TRUE;
    ELSE 
        UDP_RX_Timeout := FALSE;
    END_IF;
END_IF;

(*
====================================================
3. 速度斜坡生成
====================================================
*)
d_t := CycleTimeMs / 1000.0;

IF TargetSpeed_kmh > SpeedReference THEN
    SpeedReference := SpeedReference + RampUpRate * d_t;
    IF SpeedReference > TargetSpeed_kmh THEN SpeedReference := TargetSpeed_kmh; END_IF;
ELSE
    SpeedReference := SpeedReference - RampDownRate * d_t;
    IF SpeedReference < TargetSpeed_kmh THEN SpeedReference := TargetSpeed_kmh; END_IF;
END_IF;


(*
====================================================
5. 转向计算与CAN下发
====================================================
*)
//测试
//Target_ReardWheelAngle := Target_ReardWheelAngle_test;
Target_ReardWheelAngleAbs := ABS(Target_ReardWheelAngle);

IF Target_ReardWheelAngle >= 0 THEN
    Dir_LR := 1;
ELSE
    Dir_LR := 2;
END_IF;

SteeringRad := Target_ReardWheelAngle * PI_const / 180.0;

RackTravel_mm := Ls_mm * SteeringRad;
SteerAngle_deg := (RackTravel_mm / Pitch_mm) * 360.0;

CAN_SES_Req_F(Tgt_StrAngle := SteerAngle_deg, Tgt_StrAngleSpd := 200, Veh_Spd := 50, Enable := 1);
CAN_SES_Req_Data_F := CAN_SES_Req_F.CanData;

CAN_SES_Req_R(Tgt_StrAngle := -SteerAngle_deg, Tgt_StrAngleSpd := 200, Veh_Spd := 50, Enable := 1);
CAN_SES_Req_Data_R := CAN_SES_Req_R.CanData;

(*
====================================================
6. Ackermann运动学正解
====================================================
*)
fbKine(v_kmh := SpeedReference, delta := ABS(SteeringRad), Dir_LR := Dir_LR);

Rr_Target_rpm := fbKine.wRR_rpm;
Rl_Target_rpm := fbKine.wRL_rpm;

(*
====================================================
7. 电机反馈读取
====================================================
*)
fbDepack_MotorStatus1_RR(RxData := GVL.GCAN212_Recive_RR_status1);
fbDepack_MotorStatus1_RL(RxData := GVL.GCAN212_Recive_RL_status1);

Rr_Actual_rpm := INT_TO_LREAL(fbDepack_MotorStatus1_RR.SpeedFdk);
Rl_Actual_rpm := INT_TO_LREAL(fbDepack_MotorStatus1_RL.SpeedFdk);

//******判断是否是倒车减速******
IsReversingAndDecelerating := FALSE;
// 判断正在后退且处于减速过程
IF (SpeedReference <= 0 ) AND   // 曾经/当前在后退
   (Rr_Actual_rpm < 0) AND                               // 实际还在明显后退
   (Rr_Target_rpm> Rr_Actual_rpm) THEN                 // 目标速度 >= 当前参考速度（向0或停止靠近）
   
    IsReversingAndDecelerating := TRUE;
END_IF;


(*
7. 误差计算 + 前馈 + PI 控制
*)
Rr_SpeedError := Rr_Target_rpm - Rr_Actual_rpm;
Rl_SpeedError := Rl_Target_rpm - Rl_Actual_rpm;

FF_Torque_RR := Rr_Target_rpm * FeedforwardGain * 0.012;
FF_Torque_RL := Rl_Target_rpm * FeedforwardGain * 0.012;

Integral_RR := Integral_RR + Rr_SpeedError * Ki;
Integral_RL := Integral_RL + Rl_SpeedError * Ki;
Integral_RR := LIMIT(-IntegralLimit, Integral_RR, IntegralLimit);
Integral_RL := LIMIT(-IntegralLimit, Integral_RL, IntegralLimit);

TotalTorque_RR := FF_Torque_RR + Kp * Rr_SpeedError + Integral_RR;
TotalTorque_RL := FF_Torque_RL + Kp * Rl_SpeedError + Integral_RL;


//倒车减速给负值力矩  否则给正力矩
IF IsReversingAndDecelerating  THEN
	TotalTorque_RR := -ABS(TotalTorque_RR);
    TotalTorque_RL := -ABS(TotalTorque_RL);
	
END_IF

(*
====================================================
9. 档位与安全制动
====================================================
*)

BrakeRequest := FALSE;
// IF Break OR UDP_RX_Timeout OR GVL.Emergency_Stop OR GVL.IsCollisionF OR GVL.IsCollisionR THEN
//     BrakeRequest := TRUE;
// END_IF;
IF Break OR GVL.Emergency_Stop OR GVL.IsCollisionF OR GVL.IsCollisionR THEN
    BrakeRequest := TRUE;
END_IF;

IF BrakeRequest THEN
    PressureValue := 60;
    Enable_Motor := FALSE;
    TorqueCmd_RR := 0;
    TorqueCmd_RL := 0;
    Integral_RR := 0.0;
    Integral_RL := 0.0;
    SpeedReference := 0.0;
ELSE
    PressureValue := 0;
    Enable_Motor := TRUE;
	TotalTorque_RR := LIMIT(MinTorque, TotalTorque_RR, MaxTorque);
    TotalTorque_RL := LIMIT(MinTorque, TotalTorque_RL, MaxTorque);
    
	TorqueCmd_RR := REAL_TO_INT(TotalTorque_RR );
 	TorqueCmd_RL := REAL_TO_INT(TotalTorque_RL );
END_IF;

(*
====================================================
11. 电机指令下发
====================================================
*)
fbMotorCmd_RR(
    CanID := 16#10FFE597,
    Gear_Cmd := RR_Shift_leavel,
    DriveMode := FALSE,
    MCU_Enable := Enable_Motor,
    TorqueCmd := TorqueCmd_RR,
    TxFrame => GVL.CAN_Motor_Cmd_RR,
    UdpTxFrame => GVL.GCAN212_Send_RR_cmd
);

fbMotorCmd_RL(
    CanID := 16#10FFE597,
    Gear_Cmd := RL_Shift_leavel,
    DriveMode := FALSE,
    MCU_Enable := Enable_Motor,
    TorqueCmd := TorqueCmd_RL,
    TxFrame => GVL.CAN_Motor_Cmd_RL,
    UdpTxFrame => GVL.GCAN212_Send_RL_cmd
);

(*
====================================================
12. 制动指令
====================================================
*)
VCU_SEB_Req_Data[0] := 6;
VCU_SEB_Req_Data[3] := PressureValue;

(*
====================================================
13. 车速反解与显示
====================================================
*)
fbInvKine(
    ActVel_RL := fbDepack_MotorStatus1_RL.SpeedFdk,
    ActVel_RR := fbDepack_MotorStatus1_RR.SpeedFdk,
    SteerAngle_FL := fbKine.deltaL,
    SteerAngle_FR := fbKine.deltaR,
    radius := fbKine.radius
);
(*
====================================================================
 14. 整车状态 CAN 回传
====================================================================
*)
CAN_CCU_Send(
    CCU_ShiftLevel_Sts        := Vehicle_ShiftLevel,
    CCU_P_Sts                 := GVL.Emergency_Stop OR GVL.Remote_Break OR Break,
    CCU_Ignition_Sts          := 1,
    CCU_Drive_Mode_Shift      := 0,

    Steering_Wheel_Direction  := TRUE,

    CCU_Steering_Wheel_Angle  := fbInvKine.delta * 4.44 * 180 / 3.1415926,
    CCU_Vehicle_Speed         := fbInvKine.VehicleSpeed,

    CCU_Drive_Mode            := 0,

    Remote_Brake              := GVL.Remote_Break,
    Emergency_Brake           := GVL.Emergency_Stop,
    SCU_Brake_Singal          := Break,

    Left_Turn_Light_Sts       := 0,
    Right_Turn_Light_Sts      := 0,

    Position_Light_Sts        := 0,
    LowBeam_Sts               := 0,

    TxFrame => CCU_CAN_Data
);

(*
====================================================================
 15. BMS 状态转发
====================================================================
*)
IF ReciveCanID = 16#444 THEN

    CAN_BMS_Send(
		RxData := ReciveCanData,
        TxData => BMS_Send_Data
    );
	YkqRxPDO0_data[0] := ReciveCanData[6];
END_IF;

YkqRxPDO0_data[1] := LREAL_TO_BYTE(fbInvKine.VehicleSpeed * 10);

END_FUNCTION_BLOCK

// Device/Application/FB_SteerPositionPID
FUNCTION_BLOCK FB_SteerPositionPID
VAR_INPUT
    deltaL_ref    : LREAL;   // 期望左前轮角度 (rad)
    deltaR_ref    : LREAL;   // 期望右前轮角度 (rad)
    dt_           : LREAL := 0.01; // 控制周期 (s)
    Kp            : LREAL := 8.0;
    Ki            : LREAL := 1.0;
    Kd            : LREAL := 0.1;
    outMax        : LREAL := 1000.0;  // 速度模式输出上限 (rpm 等)
    outMin        : LREAL := -1000.0;
    derivTau      : LREAL := 0.02;
    usePositionSetpoint : BOOL := TRUE; // TRUE: 下发位置 setpoint(TRUE：位置模式； FALSE：速度模式)
    PosUnitPerRad : LREAL := 180.0/3.14159265358979323846; // 默认 deg/rad，若你的驱动用 counts 把这里改为 counts_per_rad
    VelUnitPerRadSecToPDO : LREAL := 60.0/(2.0*3.14159265358979323846); // rad/s -> rpm
END_VAR

VAR_IN_OUT
    ActPos_FL     : DINT;   // 
    ActPos_FR     : DINT;   // 
END_VAR

VAR_OUTPUT
    PDO_TargetPos_FL : DINT; //
    PDO_TargetPos_FR : DINT;
    PDO_TargetVel_FL : DINT; // 
    PDO_TargetVel_FR : DINT;
END_VAR

VAR
    actPosRadL   : LREAL;
    actPosRadR   : LREAL;
    errL, errR   : LREAL;
    prevErrL     : LREAL := 0.0;
    prevErrR     : LREAL := 0.0;
    integralL    : LREAL := 0.0;
    integralR    : LREAL := 0.0;
    derivL_filt  : LREAL := 0.0;
    derivR_filt  : LREAL := 0.0;
    alpha        : LREAL;
    deriv_rawL   : LREAL;
    deriv_rawR   : LREAL;
    pidOutL      : LREAL; // 若输出速度则单位为 rad/s (需乘 conversion)
    pidOutR      : LREAL;
    PI_CONST     : LREAL := 3.14159265358979323846;
END_VAR

IF dt_ <= 0.0 THEN dt_ := 0.01; END_IF
alpha := derivTau / (derivTau + dt_);

(* 将 ActPos (DINT, PDO units) 转为弧度 *)
actPosRadL := DINT_TO_LREAL(ActPos_FL) / PosUnitPerRad; 
actPosRadR := DINT_TO_LREAL(ActPos_FR) / PosUnitPerRad; 

(* 位置环 PID（rad 域） *)
errL := deltaL_ref - actPosRadL;
integralL := integralL + errL * dt_;
deriv_rawL := (errL - prevErrL) / dt_;
derivL_filt := alpha * derivL_filt + (1.0 - alpha) * deriv_rawL;
pidOutL := Kp * errL + Ki * integralL + Kd * derivL_filt;

IF pidOutL > outMax THEN
    pidOutL := outMax;
    integralL := integralL - errL * dt_;
ELSIF pidOutL < outMin THEN
    pidOutL := outMin;
    integralL := integralL - errL * dt_;
END_IF
prevErrL := errL;

errR := deltaR_ref - actPosRadR;
integralR := integralR + errR * dt_;
deriv_rawR := (errR - prevErrR) / dt_;
derivR_filt := alpha * derivR_filt + (1.0 - alpha) * deriv_rawR;
pidOutR := Kp * errR + Ki * integralR + Kd * derivR_filt;

IF pidOutR > outMax THEN
    pidOutR := outMax;
    integralR := integralR - errR * dt_;
ELSIF pidOutR < outMin THEN
    pidOutR := outMin;
    integralR := integralR - errR * dt_;
END_IF
prevErrR := errR;

(* 输出 *)
IF usePositionSetpoint THEN
    (* 位置模式：把目标角（rad）转换为 PDO 单位 (PosUnitPerRad)，然后 LREAL->DINT *)
    PDO_TargetPos_FL := LREAL_TO_DINT( deltaL_ref * PosUnitPerRad );  
    PDO_TargetPos_FR := LREAL_TO_DINT( deltaR_ref * PosUnitPerRad );  
    PDO_TargetVel_FL := 0;
    PDO_TargetVel_FR := 0;
ELSE
    (* 速度模式：把 pidOut (rad/s) 转换为 PDO 速度单位 (rpm) *)
    (* 先把 pidOut（rad/s）乘以系数转换为 rpm，再 LREAL->DINT *)
    PDO_TargetVel_FL := LREAL_TO_DINT( pidOutL * VelUnitPerRadSecToPDO ); 
    PDO_TargetVel_FR := LREAL_TO_DINT( pidOutR * VelUnitPerRadSecToPDO ); 
    PDO_TargetPos_FL := 0;
    PDO_TargetPos_FR := 0;
END_IF

END_FUNCTION_BLOCK

// Device/Application/FB_RearWheelVelocityPID
FUNCTION_BLOCK FB_RearWheelVelocityPID
VAR_INPUT
    omegaRL_ref   : LREAL;   // 左后轮目标角速 (rad/s)
    omegaRR_ref   : LREAL;   // 右后轮目标角速 (rad/s)
    dt_           : LREAL := 0.01;
    Kp            : LREAL := 5;
    Ki            : LREAL := 0;
    Kd            : LREAL := 0;
    outMax        : LREAL := 3000.0;  // 最大输出(rpm)，调为合适值
    outMin        : LREAL := -3000.0;
    derivTau      : LREAL := 0.02;
END_VAR

VAR_IN_OUT
    ActVel_RL     : DINT;   // <<< 修改：来自 PDO 反馈 (rpm) (DINT)
    ActVel_RR     : DINT;   // <<< 修改：来自 PDO 反馈 (rpm) (DINT)
END_VAR

VAR_OUTPUT
    PDO_TargetVel_RL : DINT; // <<< 修改：下发给驱动 (rpm) (DINT)
    PDO_TargetVel_RR : DINT; // <<< 修改
END_VAR

VAR
    (* 内部以 LREAL 进行 PID 运算，单位为 rpm *)
    rpmRefRL      : LREAL;
    rpmRefRR      : LREAL;
    actRPM_RL     : LREAL;
    actRPM_RR     : LREAL;
    errRL, errRR  : LREAL;
    prevErrRL     : LREAL := 0.0;
    prevErrRR     : LREAL := 0.0;
    integralRL    : LREAL := 0.0;
    integralRR    : LREAL := 0.0;
    derivFiltRL   : LREAL := 0.0;
    derivFiltRR   : LREAL := 0.0;
    alpha         : LREAL;
    deriv_rawRL   : LREAL;
    deriv_rawRR   : LREAL;
    pidOutRL      : LREAL;
    pidOutRR      : LREAL;
    u_raw_RL      : LREAL;
    u_raw_RR      : LREAL;
    u_cmd_RL      : LREAL;
    u_cmd_RR      : LREAL;
    PI_CONST      : LREAL := 3.14159265358979323846;
    convVel       : LREAL; // 转换系数：rad/s -> rpm = 60/(2*pi)
END_VAR

(* 保护 *)
IF dt_ <= 0.0 THEN dt_ := 0.01; END_IF
alpha := derivTau / (derivTau + dt_);
convVel := 60.0 / (2.0 * PI_CONST); // rad/s -> rpm

(* 1) 参考角速 rad/s -> rpm *)
rpmRefRL := omegaRL_ref * convVel;   // LREAL
rpmRefRR := omegaRR_ref * convVel;

(* 2) 反馈 DINT -> LREAL (rpm) *)
actRPM_RL := DINT_TO_LREAL(ActVel_RL);       // <<< 修改：显式转换 DINT -> LREAL
actRPM_RR := DINT_TO_LREAL(ActVel_RR);       // <<< 修改

(* 左轮 PID（单位：rpm） *)
errRL := rpmRefRL - actRPM_RL;                       // 目标 - 实测 (rpm)
integralRL := integralRL + errRL * dt_;
deriv_rawRL := (errRL - prevErrRL) / dt_;
derivFiltRL := alpha * derivFiltRL + (1.0 - alpha) * deriv_rawRL;
pidOutRL := Kp * errRL + Ki * integralRL + Kd * derivFiltRL;

(* 抗饱和：若 pidOut 超限则回退积分 *)
u_raw_RL := rpmRefRL + pidOutRL;   // 运动学前馈 + PID 修正 (rpm)
IF u_raw_RL > outMax THEN
    u_cmd_RL := outMax;
ELSIF u_raw_RL < outMin THEN
    u_cmd_RL := outMin;
ELSE
    u_cmd_RL := u_raw_RL;
END_IF

(* 选用简单抗积分风up：当饱和且误差驱动方向使积分继续发散时回退积分 *)
IF (u_cmd_RL <> u_raw_RL) THEN
    (* 饱和，做积分回退 *)
    integralRL := integralRL - errRL * dt_;
END_IF

prevErrRL := errRL;

(* 右轮 PID（单位：rpm） *)
errRR := rpmRefRR - actRPM_RR;
integralRR := integralRR + errRR * dt_;
deriv_rawRR := (errRR - prevErrRR) / dt_;
derivFiltRR := alpha * derivFiltRR + (1.0 - alpha) * deriv_rawRR;
pidOutRR := Kp * errRR + Ki * integralRR + Kd * derivFiltRR;

u_raw_RR := rpmRefRR + pidOutRR;
IF u_raw_RR > outMax THEN
    u_cmd_RR := outMax;
ELSIF u_raw_RR < outMin THEN
    u_cmd_RR := outMin;
ELSE
    u_cmd_RR := u_raw_RR;
END_IF

IF (u_cmd_RR <> u_raw_RR) THEN
    integralRR := integralRR - errRR * dt_;
END_IF

prevErrRR := errRR;

(* 3) 输出：转换为 DINT 并下发到 PDO (rpm) *)
(* 注意：DINT(...) 有截断行为，请确保 outMax/outMin 在 DINT 可表示范围内 *)
PDO_TargetVel_RL := LREAL_TO_DINT(u_cmd_RL);  // <<< 修改：显式转换为 DINT
PDO_TargetVel_RR := LREAL_TO_DINT(u_cmd_RR);  // <<< 修改

// IF PDO_TargetVel_RL > GVL.MaxMotorSpeed THEN
// 	PDO_TargetVel_RL := GVL.MaxMotorSpeed;
// END_IF
// 
// IF PDO_TargetVel_RR > GVL.MaxMotorSpeed THEN
// 	PDO_TargetVel_RR := GVL.MaxMotorSpeed;
// END_IF

END_FUNCTION_BLOCK

// Device/Application/FB_CAN_VCU_SES_Req
FUNCTION_BLOCK FB_CAN_VCU_SES_Req
VAR_INPUT
    Tgt_StrAngle      : REAL;   // 目标转向角（°）
    Tgt_StrAngleSpd   : REAL;   // 目标转向角速度（°/s）
    Veh_Spd           : BYTE;   // 车速（可选，直接填 Byte6）
    Enable            : BOOL;   // 角度控制使能
END_VAR

VAR_OUTPUT
    CanData : ARRAY[0..7] OF BYTE; // 最终 8 字节 CAN 数据
END_VAR

VAR
    RawAngle   : UINT;   // 16bit 原始角度
    RawSpd     : UINT;   // 16bit 原始角速度
    RollCnt    : BYTE;   // 4bit Rolling Counter
    Sum        : UINT;
    i          : INT;
END_VAR

//============================================================
// 1. 物理量 → 原始值
//============================================================

// 角度：Phys = Raw*0.1 - 3000
RawAngle := REAL_TO_UINT((Tgt_StrAngle + 3000.0) / 0.1);

// 角速度：1 °/s per bit
RawSpd := REAL_TO_UINT(Tgt_StrAngleSpd);

//============================================================
// 2. 清空数据
//============================================================
FOR i := 0 TO 7 DO
    CanData[i] := 0;
END_FOR;

//============================================================
// 3. Byte0：控制位
// bit1 = AngleControl_Enable
// bit0 = Alignment_Enable（这里不用，置0）
//============================================================
IF Enable THEN
    CanData[0] := 2;   // 0000 0010
ELSE
    CanData[0] := 0;
END_IF;

//============================================================
// 4. 转向角（Motorola）
// 高字节 → Byte1
// 低字节 → Byte2
//============================================================
CanData[1] := UINT_TO_BYTE(SHR(RawAngle, 8));
CanData[2] := UINT_TO_BYTE(RawAngle AND 16#FF);

//============================================================
// 5. 转向角速度（Motorola）
// 高字节 → Byte3
// 低字节 → Byte4
//============================================================
CanData[3] := UINT_TO_BYTE(SHR(RawSpd, 8));
CanData[4] := UINT_TO_BYTE(RawSpd AND 16#FF);

//============================================================
// 6. Byte5：Rolling Counter + Enable
// bit0 = RollCnt_Enable
// bit1 = CheckSum_Enable
// bit4~7 = Rolling Counter
//============================================================
CanData[5] := 16#03 OR SHL(RollCnt AND 16#0F, 4);

//============================================================
// 7. Byte6：车速
//============================================================
CanData[6] := Veh_Spd;

//============================================================
// 8. Checksum
// CheckSum = (Byte0 + ... + Byte6) XOR 0xFF
//============================================================
Sum := 0;
FOR i := 0 TO 6 DO
    Sum := Sum + CanData[i];
END_FOR;

CanData[7] := UINT_TO_BYTE((Sum AND 16#FF) XOR 16#FF);

//============================================================
// 9. Rolling Counter 自增
//============================================================
RollCnt := (RollCnt + 1) AND 16#0F;

END_FUNCTION_BLOCK

// Device/Application/cantesttest
FUNCTION_BLOCK cantesttest
VAR_INPUT
END_VAR
VAR_OUTPUT
END_VAR
VAR
	CANBus_CtrlDevState_0: CANBus_CtrlDevState;
	cmd: CANBus_CtrlCmdType_Enum;
	exc: BOOL;
	CANBus_DevRxMsg_0: CANBus_DevRxMsg;
	rxfilter: CANBus_RxFilter_t;
	RxMsg: CANBus_FrameMsg_t;
END_VAR

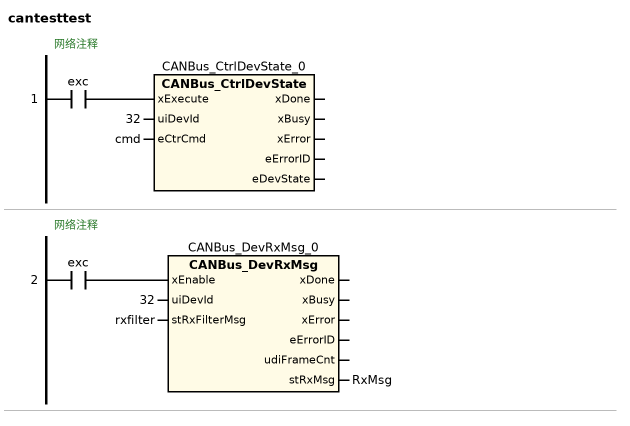
// NETWORK 1
// 网络注释
CANBus_CtrlDevState_0(xExecute := exc, uiDevId := 32, eCtrCmd := cmd); // CANBus_CtrlDevState

// NETWORK 2
// 网络注释
CANBus_DevRxMsg_0(xEnable := exc, uiDevId := 32, stRxFilterMsg := rxfilter, stRxMsg => RxMsg); // CANBus_DevRxMsg

END_FUNCTION_BLOCK
